# B&R Automation Studio project Parker_BMM_ST_V5_3147_V12 (part 17)

#### cur_draw.c
```c
/********************************************************************
 * COPYRIGHT --  B&R CHINA
 ********************************************************************
 * Program: cur_draw
 * File: cur_draw.c
 * Author: lijianjun
 * Created: March 06, 2013
 ********************************************************************
 * Implementation of program cur_draw --- thick profile curve draw in HMI
 ********************************************************************/

#include <bur/plctypes.h>
#include <string.h>

#ifdef _DEFAULT_INCLUDES
#include <AsDefault.h>
#endif

/***********************************************************************************
** 			                    Include user files								  **
***********************************************************************************/
#include "draw.h"
#include "pic_id.h"
#include "thick.h"

/***********************************************************************************
                             Function Declarations
***********************************************************************************/
UINT vsLine( UDINT VCHandle, UINT x1, UINT y1,UINT x2, UINT y2, USINT color);
UINT vsLineH( UDINT VCHandle, UINT x, UINT y, UINT len, USINT color);
UINT vsLineV( UDINT VCHandle, UINT x, UINT y, UINT len, USINT color);
UINT vsRect(  UDINT VCHandle, UINT x1, UINT y1,UINT x2, UINT y2, USINT color);

/**********************************************************************************
**     	        		 I N I T U P  O F   T H E   T A S K 		 		     **
**********************************************************************************/
_INIT  void init(void)
{
	width 		= 	VSCREEN_WIDTH;
	height 		= 	VSCREEN_HEIGHT;
	backColor  	= 	VSCREEN_COLOR_BACKGROUND;
	frameColor 	= 	VSCREEN_COLOR_FRAME;
	crossColor	= 	VSCREEN_COLOR_CROSS_CURSOR;
	fillColor   =  VSCREEN_COLOR_BACKGROUND;

	ORIGINAL_X0  = 100;
	ORIGINAL_Y0  = 150;

	rSetScale = 0.1;
	rActScale = 1.0;
	xScaleBmp = 0;

	drawStep = 0;
}/*  end of INIT */

/**********************************************************************************
**        	     C Y C L I C   P A R T   O F   T H E   T A S K  				 **
**********************************************************************************/
_CYCLIC void cyc(void)
{
	INT X,Y;

	if((gPanelObj.GetPicture == PIC_CURVE_TRACE) ||
		(1 == gThickProf.FunOption.IsTraceInEdit && gPanelObj.GetPicture == PIC_CURVE_EDIT))
	{
		if (memcmp(getAT,gThickData.RealData,sizeof(getAT)) != 0 && DrawMan.draw == 0)
		{
			DrawMan.draw = 1;
			memcpy(getAT,gThickData.RealData,sizeof(getAT));
		}
	}

	if (gPanelObj.GetPicture == PIC_CURVE_EDIT)
	{
		if (DRAW_PIC != PIC_CURVE_EDIT && DRAW_PIC != 255)
		{
			DrawMan.draw = 1;
		}
		DRAW_PIC = PIC_CURVE_EDIT;
	}
	else if (gPanelObj.GetPicture == PIC_CURVE_TRACE)
	{
		if (DRAW_PIC != PIC_CURVE_TRACE && DRAW_PIC != 255)
		{
			DrawMan.draw = 1;
		}
		DRAW_PIC = PIC_CURVE_TRACE;
	}
	else
	{
		DRAW_PIC = 255;
	}

	if (gPanelObj.GetPicture == PIC_CURVE_EDIT || gPanelObj.GetPicture == PIC_CURVE_TRACE)
	{
		switch (drawStep)
		{
			case 0:
				vcHandle = VA_Setup(1,gPanelObj.VisualName);
				if (vcHandle)  drawStep = 100;
				break;

			case 100:
				status = VA_Saccess(1, vcHandle);
				if(status == 0)
				{
					drawStep = 200;
				}
				break;

			case 200:
				Status_Attach = 1;
				if (gPanelObj.GetPicture == PIC_CURVE_EDIT)
				{
					Status_Attach = VA_Attach(1,vcHandle,0,(UDINT)"Page_82_Profile/Default/DrawBox_1");
				}
				else
				{
					Status_Attach = VA_Attach(1,vcHandle,0,(UDINT)"Page_83_Trace/Default/DrawBox_1");
				}
				if(Status_Attach == 0)
				{
					/* Get width of DrawBox Control*/
					VA_GetDisplayInfo(1,vcHandle,1,(UDINT)&Drawbox_width);
					/* Get height of DrawBox Control */
					VA_GetDisplayInfo(1,vcHandle,2,(UDINT)&Drawbox_height);

					drawStep = 300;
				}
				else
				{
					VA_Srelease(1, vcHandle);
					drawStep = 100;
				}
				break;
			case 300:
				xMax = 0.0;
				for(i=0;i<= S$THICK_MAX;i++)
					{
					if(xMax < SetPos[i].x)xMax = SetPos[i].x;
				}

				if (usScaleIndex == 1) //ipis0619
				{
					rSetScale = 0.4;
					rActScale = 4.0;
					xScaleBmp = 2;
				}else if (usScaleIndex == 2)
				{
					rSetScale = 0.2;
					rActScale = 2.0;
					xScaleBmp = 1;
				}else
				{
					rSetScale = 0.1;
					rActScale = 1.0;
					xScaleBmp = 0;
				}
		/*---//ipis0619 -----------------------------------------*/
//				if(xMax >= 1500)
//				{
//					rSetScale = 0.1;
//					rActScale = 1.0;
//					xScaleBmp = 0;
//				}
//				else if(xMax >= 750)
//				{
//					rSetScale = 0.2;
//					rActScale = 2.0;
//					xScaleBmp = 1;
//				}
//				else
//				{
//					rSetScale = 0.4;
//					rActScale = 4.0;
//					xScaleBmp = 2;
//				}
		/*---//ipis0619 -----------------------------------------*/
				status = VA_Redraw (1,vcHandle);
				if(0 == status)
				{
					if (gPanelObj.GetPicture == PIC_CURVE_EDIT)  drawStep  = 400;
					if (gPanelObj.GetPicture == PIC_CURVE_TRACE) drawStep  = 600;
				}
				break;
			/**************draw the setting curve*************/
			case 400:
				for(i=0;i<= S$THICK_MAX;i++)
					{
					X = (INT)(SetPos[i].x*rSetScale + 0.1);
					if(X > Drawbox_width - 2)X = Drawbox_width - 2;
					Y = S$THICK_POINT - SetPos[i].y;    /* 0 <SetPos[i].y <= 399  ->  1 < Y < 400*/

					vsLineH(vcHandle,0,Y,Drawbox_width-1,VSCREEN_COLOR_BACKGROUND);

					if (1 == CurveNode[i].flagNode)
					{
						if(i == DrawMan.currentNode && 1 == DrawMan.flagLineFocus)
						{
							vsLineH(vcHandle,0,Y,X,crossColor);
							vsLineH(vcHandle,0,Y,DrawMan.weight*rSetScale,VSCREEN_COLOR_WEIGHT);
						}
						else
						{
							vsLineH(vcHandle,0,Y,X,VSCREEN_COLOR_CURVE);
							vsLineH(vcHandle,0,Y,DrawMan.weight*rSetScale,VSCREEN_COLOR_WEIGHT);
						}
					}
					else
					{
						vsLineH(vcHandle,0,Y,X,VSCREEN_COLOR_UNFOCUS_LINE);
						vsLineH(vcHandle,0,Y,DrawMan.weight*rSetScale,VSCREEN_COLOR_WEIGHT);
					}

					if(0 == DrawMan.flagLineFocus)
					{
						if(i > CurveNode[DrawMan.currentNode].former + 1 && i <= DrawMan.currentNode)
						{
							vsLine(vcHandle,(INT)(SetPos[i-1].x*rSetScale + 0.1),S$THICK_POINT - SetPos[i-1].y,X,Y,crossColor);
								}
						else
						{
							if(i > 0)
							{
								vsLine(vcHandle,(INT)(SetPos[i-1].x*rSetScale + 0.1),S$THICK_POINT - SetPos[i-1].y,X,Y,VSCREEN_COLOR_CURVE);
									}
						}
					}
					else
					{
						if(i > 0)
						{
							vsLine(vcHandle,(INT)(SetPos[i-1].x*rSetScale + 0.1),S$THICK_POINT - SetPos[i-1].y,X,Y,VSCREEN_COLOR_CURVE);
								}
					}
				}

				if(DrawMan.step == S$STEP_ADDLINE)
					{
					drawStep = 500;
				}
				else
				{
					drawStep = 550;
				}
				break;
			/*---draw the cross line ---*/
			case 500:
				xTemp = (INT)(SetPos[DrawMan.currentPoint].x*rSetScale + 0.1) - 20;
				if(xTemp < 0)xTemp = 0;

				if(xTemp + 40 < width)
				{
					xLength = 40;
				}
				else
				{
					xLength = width - 40;
				}
				vsLineH(vcHandle,xTemp,S$THICK_POINT - DrawMan.currentPoint,xLength,crossColor);

					yTemp	= S$THICK_POINT - DrawMan.currentPoint - 20;
				if(yTemp < 0)yTemp = 0;

				if(yTemp + 40 < height)
				{
					yLength = 40;
				}
				else
				{
					yLength = height - 40;
				}
				vsLineV(vcHandle,(INT)(SetPos[DrawMan.currentPoint].x*rSetScale + 0.1),yTemp,yLength,crossColor);
				drawStep = 550;
				break;
			/*------ is or not draw the trace curve in edit profile page ------*/
			case 550:
				if(1 == gThickProf.FunOption.IsTraceInEdit)
				{
					drawStep = 700;
				}
				else
				{
					drawStep = 900;
				}
				break;
			/**************draw the setting curve*************/
			case 600:
				for(i=0;i<= S$THICK_MAX;i++)
					{
					vsLineH(vcHandle,0,S$THICK_POINT - SetPos[i].y,Drawbox_width-1,VSCREEN_COLOR_BACKGROUND);
						vsLineH(vcHandle,0,S$THICK_POINT - SetPos[i].y,(INT)(SetPos[i].x*rSetScale + 0.1),VSCREEN_COLOR_UNFOCUS_LINE);
						}
				drawStep = 700;
				break;
			/**************draw the trace curve*************/
			case 700:
				for(i=0;i<S$THICK_SAMPLE-1;i++)
					{
					if (getAT[i+1] != 0)
					{
						firstPos.x  = getAT[i] * rActScale;
						firstPos.y  = i*4;
						secondPos.x = getAT[i+1] * rActScale;
						secondPos.y = (i+1)*4;
						status = vsLine(vcHandle, firstPos.x, S$THICK_POINT-firstPos.y, secondPos.x, S$THICK_POINT-secondPos.y, crossColor);
							}
				}

				if(getAT[S$THICK_SAMPLE-1]!= 0)
					{
					status = vsLine(vcHandle, getAT[S$THICK_SAMPLE-1] * rActScale, S$THICK_POINT - 396, getAT[S$THICK_SAMPLE-1] * rActScale, S$THICK_POINT - 399, crossColor);
						}
				drawStep = 900;
				break;
			/* copy the screen to interface  */
			case 900:
				vsRect(vcHandle,0,0,VSCREEN_WIDTH-1,VSCREEN_HEIGHT-1,VSCREEN_COLOR_FRAME);
				VA_Redraw (1,vcHandle);
				VA_Detach(1,vcHandle);
				VA_Srelease(1, vcHandle);
				if((gPanelObj.GetPicture == PIC_CURVE_EDIT) || (gPanelObj.GetPicture == PIC_CURVE_TRACE))
				{
					DrawMan.draw = 0;
					drawStep = 1000;
				}
				else
				{
					drawStep = 2000;
				}
				break;
			/*	waiting for draw  */
			case 1000:
				if (1 == DrawMan.draw )
				{
					drawStep  = 100;
				}
				break;
			case 2000:
				drawStep  = 100;
				break;
		}
	}
	else
	{
		if (drawStep != 0 && vcHandle != 0) drawStep = 100;
	}

}/*end of CYCLIC*/

UINT vsLine( UDINT VCHandle, UINT x1, UINT y1,UINT x2, UINT y2, USINT color)
{
	if(x1 > Drawbox_width-2)x1 = Drawbox_width-2;
	if(x2 > Drawbox_width-2)x2 = Drawbox_width-2;
	return  VA_Line(1, VCHandle,x1,y1,x2,y2,color);
}

UINT vsLineH( UDINT VCHandle, UINT x, UINT y, UINT len, USINT color)
{
	if(x+len <= Drawbox_width-2)
	{
		return  VA_Line(1, VCHandle,x,y,x+len,y,color);
	}
	else
	{
		return  VA_Line(1, VCHandle,x,y,Drawbox_width-2,y,color);
	}
}

UINT vsLineV( UDINT VCHandle, UINT x, UINT y, UINT len, USINT color)
{
	if(x > Drawbox_width-2)x = Drawbox_width-2;
	return  VA_Line(1, VCHandle,x,y,x,y+len,color);
}

UINT vsRect(  UDINT VCHandle, UINT x1, UINT y1,UINT x2, UINT y2, USINT color)
{
	return VA_Rect(1,VCHandle,x1,y1,x2-x1,y2-y1,255,color);
}
```

#### cur_draw.var
```iecst
VAR
	vcHandle : UDINT;
	xTemp : INT;
	xLength : INT;
	yTemp : INT;
	yLength : INT;
	width : UINT;
	Drawbox_width : UDINT;
	Drawbox_height : UDINT;
	height : UINT;
	backColor : UINT;
	fillColor : UINT;
	frameColor : UINT;
	crossColor : UINT;
	xMax : INT;
	xScaleBmp : UINT;
	rSetScale : REAL;
	rActScale : REAL;
	status : UINT;
	Status_Attach : UINT;
	drawStep : UINT;
	i : UINT;
	getAT : ARRAY[0..99] OF INT;
	DRAW_PIC : UINT;
	firstPos : position_typ;
	secondPos : position_typ;
END_VAR
```

### Program Logical/thickness/cur_edit (ANSIC, version 1.00.0) - profile edit

#### cur_edit.c
```c
/********************************************************************
 * COPYRIGHT --  B&R CHINA
 ********************************************************************
 * Program: cur_edit
 * File: cur_edit.c
 * Author: lijianjun
 * Created: March 06, 2013
 ********************************************************************
 * Implementation of program cur_edit --- thick profile curve data compiling
 ********************************************************************/

#include <bur/plctypes.h>
#include <string.h>

#ifdef _DEFAULT_INCLUDES
#include <AsDefault.h>
#endif

/***********************************************************************************
** 					 	        Include user files								             **
***********************************************************************************/
#include "keyap2100.h"
#include "pic_id.h"
#include "draw.h"
#include "thick.h"
#include "edge.h"               /*edge function
/**********************************************************************************
**                            Function Declarations								      **
**********************************************************************************/
void nodeAdd(USINT *enable,UINT nodeNum); /*insert a horizontal line*/
void nodeDel(USINT *enable,UINT nodeNum); /*delete a horizontal line*/
void curveScan(SINT *upDown);  			   /*scan the horizontal to get the focus*/
void curveQuickScan(SINT *upDown);  		/*scan the horizontal to get the focus*/
void curveColor(USINT *action);			   /* */
void vxEdit();
void vxEditUnit(INT unitLength);
void moveCross(SINT *upDown);
void weightSet();
void curveToLine(USINT *action,UINT nodeNum);
void curveMove();
void curveClear();
/**********************************************************************************
**     	        	 I N I T U P  O F   T H E   T A S K 		 				 **
**********************************************************************************/
_INIT  void init(void)
{
	RTInfo_v.enable = 1;
	RTInfo(&RTInfo_v);
	TimeLenth = RTInfo_v.cycle_time/4000;
	tTask = RTInfo_v.cycle_time/1000.0/1000.0;

	TimeLenth  = TimeLenth /6 * 6;
	StepLength = TimeLenth;

	focusColor 		= VSCREEN_COLOR_FOCUS_LINE;
	unfocusColor 	= VSCREEN_COLOR_UNFOCUS_LINE;

	addNode 		= 0;
	delNode 		= 0;
	scanNode  	= 0;
	scanLine    = 0;
	setColor		= 0;
	isDownLoad  = 0;

	memset(oldSetPos,0,sizeof(oldSetPos));
	DrawMan.step  = S$STEP_EDIT;
	DrawMan.input = 0;

	Counter = 0;
	CurevInitDownload = 1;

	moveValue = 0;
	bBackEnable = 0;
	bRedoEnable = 0;

	memset(&gThickProf.IsMarker[0],0,sizeof(gThickProf.IsMarker));
	memset(&IsMarkerOld[0],0,sizeof(IsMarkerOld));

	MarkPercentOld = MarkPercent = 20;

	bStartUpLineFocus = 0;
	bStartDnLineFocus = 0;
	cntUpButtonPress = 0;
	cntDownButtonPress = 0;
}/*  end of init   */
/**********************************************************************************
**            C Y C L I C   P A R T   O F   T H E   T A S K  				     **
**********************************************************************************/
_CYCLIC void cyc(void)
{
	if(1 == gRecipeOperate.OnceOk && 1 == gRecipeOperate.CurveOk)
	{
		if(1 == CurevInitDownload)
		{
			CurevInitDownload = 0;
			DrawMan.downLoad  = 1;
		}

		if(1 == GapMaxLimitChange)
		{
			GapMaxLimitChange = 0;
			DrawMan.downLoad  = 1;
		}
	}

	/*IsZeroDn Change */
	if(IsZeroDnOld != gThickProf.FunOption.IsZeroDn)
	{
		DrawMan.downLoad = 1;
	}

	IsZeroDnOld = gThickProf.FunOption.IsZeroDn;

	/*  mark point --- display  */
	if((PIC_MARKER_SET_A == GetPictureOld) && (gPanelObj.GetPicture != PIC_MARKER_SET_A))
	{
		memset(&gThickProf.IsMarker[0],0,sizeof(gThickProf.IsMarker));
		memset(&IsMarkerOld[0],0,sizeof(IsMarkerOld));
		DrawMan.downLoad = 1;
	}
	GetPictureOld = gPanelObj.GetPicture;

	if(MarkPercent < -50 || MarkPercent > 50)MarkPercent = 20;
	if(MarkPercentOld != MarkPercent)
	{
		DrawMan.downLoad = 1;
	}
	MarkPercentOld = MarkPercent;

	if (memcmp(gThickProf.IsMarker,IsMarkerOld,sizeof(IsMarkerOld)) != 0)
	{
		memcpy(IsMarkerOld,gThickProf.IsMarker,sizeof(gThickProf.IsMarker));
		DrawMan.downLoad = 1;
	}

	if(ServoMinOld != gThickData.ServoMin)
	{
		isDownLoad = 2;
	}

	ServoMinOld = gThickData.ServoMin;

	if(ServoMaxOld != gThickData.ServoMax)
	{
		isDownLoad = 2;
	}

	ServoMaxOld = gThickData.ServoMax;

	if (1 == DrawMan.downLoad)
	{
		for (i = 0; i< 100; i++)
		{
			if(gMachineFix.Parison.eActuatorType == ACTUATOR_ELECTRIC  || 0 == gThickData.IsZeroDn)
			{
				gThickData.SetData[i] = gThickData.ServoMin + gThickData.ServoLength * (SetPos[i*4].x +
					SetPos[i*4+1].x + SetPos[i*4+2].x + SetPos[i*4+3].x)/12000;

				if(1 == gThickProf.IsMarker[i])
				{
					if(0 == i)
					{
						gThickData.SetData[i] = gThickData.SetData[i] + gThickData.ServoLength * MarkPercent / 100;
						if(gThickData.SetData[i] < gThickData.ServoMin)gThickData.SetData[i] = gThickData.ServoMin;
						if(gThickData.SetData[i] > gThickData.ServoMax)gThickData.SetData[i] = gThickData.ServoMax;

						gThickData.SetData[i+1] = gThickData.SetData[i+1] + gThickData.ServoLength * MarkPercent / 200;
						if(gThickData.SetData[i+1] < gThickData.ServoMin)gThickData.SetData[i+1] = gThickData.ServoMin;
						if(gThickData.SetData[i+1] > gThickData.ServoMax)gThickData.SetData[i+1] = gThickData.ServoMax;

					}
					else if(99 == i)
					{
						gThickData.SetData[i-1] = gThickData.SetData[i-1] + gThickData.ServoLength * MarkPercent / 200;
						if(gThickData.SetData[i-1] < gThickData.ServoMin)gThickData.SetData[i-1] = gThickData.ServoMin;
						if(gThickData.SetData[i-1] > gThickData.ServoMax)gThickData.SetData[i-1] = gThickData.ServoMax;

						gThickData.SetData[i] = gThickData.SetData[i] + gThickData.ServoLength * MarkPercent / 100;
						if(gThickData.SetData[i] < gThickData.ServoMin)gThickData.SetData[i] = gThickData.ServoMin;
						if(gThickData.SetData[i] > gThickData.ServoMax)gThickData.SetData[i] = gThickData.ServoMax;
					}
					else
					{
						gThickData.SetData[i-1] = gThickData.SetData[i-1] + gThickData.ServoLength * MarkPercent / 200;
						if(gThickData.SetData[i-1] < gThickData.ServoMin)gThickData.SetData[i-1] = gThickData.ServoMin;
						if(gThickData.SetData[i-1] > gThickData.ServoMax)gThickData.SetData[i-1] = gThickData.ServoMax;

						gThickData.SetData[i] = gThickData.SetData[i] + gThickData.ServoLength * MarkPercent / 100;
						if(gThickData.SetData[i] < gThickData.ServoMin)gThickData.SetData[i] = gThickData.ServoMin;
						if(gThickData.SetData[i] > gThickData.ServoMax)gThickData.SetData[i] = gThickData.ServoMax;

						gThickData.SetData[i+1] = gThickData.SetData[i+1] + gThickData.ServoLength * MarkPercent / 200;
						if(gThickData.SetData[i+1] < gThickData.ServoMin)gThickData.SetData[i+1] = gThickData.ServoMin;
						if(gThickData.SetData[i+1] > gThickData.ServoMax)gThickData.SetData[i+1] = gThickData.ServoMax;
					}
				}
			}
			else if( gMachineFix.Parison.eActuatorType == ACTUATOR_HYD && 1 == gThickData.IsZeroDn)
			{
				gThickData.SetData[i] = gThickData.ServoMax - gThickData.ServoLength * (SetPos[i*4].x +
					SetPos[i*4+1].x + SetPos[i*4+2].x + + SetPos[i*4+3].x)/12000;

				if(1 == gThickProf.IsMarker[i])
				{
					if(0 == i)
					{
						gThickData.SetData[i] = gThickData.SetData[i] - gThickData.ServoLength * MarkPercent / 100;
						if(gThickData.SetData[i] < gThickData.ServoMin)gThickData.SetData[i] = gThickData.ServoMin;
						if(gThickData.SetData[i] > gThickData.ServoMax)gThickData.SetData[i] = gThickData.ServoMax;

						gThickData.SetData[i+1] = gThickData.SetData[i+1] - gThickData.ServoLength * MarkPercent / 200;
						if(gThickData.SetData[i+1] < gThickData.ServoMin)gThickData.SetData[i+1] = gThickData.ServoMin;
						if(gThickData.SetData[i+1] > gThickData.ServoMax)gThickData.SetData[i+1] = gThickData.ServoMax;
					}
					else if(99 == i)
					{
						gThickData.SetData[i-1] = gThickData.SetData[i-1] - gThickData.ServoLength * MarkPercent / 200;
						if(gThickData.SetData[i-1] < gThickData.ServoMin)gThickData.SetData[i-1] = gThickData.ServoMin;
						if(gThickData.SetData[i-1] > gThickData.ServoMax)gThickData.SetData[i-1] = gThickData.ServoMax;

						gThickData.SetData[i] = gThickData.SetData[i] - gThickData.ServoLength * MarkPercent / 100;
						if(gThickData.SetData[i] < gThickData.ServoMin)gThickData.SetData[i] = gThickData.ServoMin;
						if(gThickData.SetData[i] > gThickData.ServoMax)gThickData.SetData[i] = gThickData.ServoMax;
					}
					else
					{
						gThickData.SetData[i-1] = gThickData.SetData[i-1] - gThickData.ServoLength * MarkPercent / 200;
						if(gThickData.SetData[i-1] < gThickData.ServoMin)gThickData.SetData[i-1] = gThickData.ServoMin;
						if(gThickData.SetData[i-1] > gThickData.ServoMax)gThickData.SetData[i-1] = gThickData.ServoMax;

						gThickData.SetData[i] = gThickData.SetData[i] - gThickData.ServoLength * MarkPercent / 100;
						if(gThickData.SetData[i] < gThickData.ServoMin)gThickData.SetData[i] = gThickData.ServoMin;
						if(gThickData.SetData[i] > gThickData.ServoMax)gThickData.SetData[i] = gThickData.ServoMax;

						gThickData.SetData[i+1] = gThickData.SetData[i+1] - gThickData.ServoLength * MarkPercent / 200;
						if(gThickData.SetData[i+1] < gThickData.ServoMin)gThickData.SetData[i+1] = gThickData.ServoMin;
						if(gThickData.SetData[i+1] > gThickData.ServoMax)gThickData.SetData[i+1] = gThickData.ServoMax;
					}
				}
			}

			x_Profile[i] = (SetPos[i*4].x + SetPos[i*4+1].x + SetPos[i*4+2].x + SetPos[i*4+3].x)/120.0;
		}

		memcpy(oldSetPos,SetPos,sizeof(SetPos));

		DrawMan.downLoad  		 = 0;
		gRecipeOperate.CurveSave = 1;
		isDownLoad        		 = 0;

	}/* if (1 == DrawMan.downLoad) */

	if(gPanelObj.GetPicture == PIC_CURVE_EDIT)
	{
		gPanelObj.LedMatric[S$KEYMATRIX_F15] =  0;
		gPanelObj.LedMatric[S$KEYMATRIX_F15] = isDownLoad;
	}
	else if(gPanelObj.GetPicture == PIC_THICK_START)
	{
		gPanelObj.LedMatric[S$KEYMATRIX_F15] = isDownLoad;
		gPanelObj.LedMatric[S$KEYMATRIX_F15] =  0;
	}
	else
	{
		gPanelObj.LedMatric[S$KEYMATRIX_F15] =  0;
		gPanelObj.LedMatric[S$KEYMATRIX_F15] =  0;
	}

	if(gPanelObj.GetPicture != PIC_CURVE_EDIT  && gPanelObj.GetPicture != PIC_THICK_START)
	{
		Counter = 0;
		return;
	}

	Counter ++;
	if(Counter > 1000)Counter = 120;
	if(Counter < 15)return;

	if(0 == gThickProf.FunOption.IsAccu)
	{
		AccuColor  = 0x0060;
		ContiColor = 0x003A;

	}
	else
	{
		AccuColor  = 0x003A;
		ContiColor = 0x0060;
	}

	if((gPanelObj.PasswordLevel >= 1)&&(1 == DrawMan.flagLineFocus)&& (DrawMan.step == S$STEP_EDIT))
	{
		inputenable = 1;
	}
	else
	{
		inputenable = 0;
	}

	bHideBack = ! bBackEnable;

	if(gPanelObj.GetPicture == PIC_CURVE_EDIT)
	{
		if(gPanelObj.PasswordLevel >= 1)
		{
			if(gPanelObj.PasswordLevel >= 3)
			{
			//	changeButton = gPanelObj.KeyMatric[S$KEYMATRIX_F7];
			}
			else
			{
				changeButton = 0;
			}
//			delButton 		= gPanelObj.KeyMatric[S$KEYMATRIX_F8] | gPanelObj.KeyMatric[S$KEYMATRIX_DEL];
//			curtolButton 	= gPanelObj.KeyMatric[S$KEYMATRIX_F9] | bCurveChangeLine;
			delButton 		=  gPanelObj.KeyMatric[S$KEYMATRIX_DEL];
			curtolButton 	=  bCurveChangeLine;
			escButton 		= gPanelObj.KeyMatric[S$KEYMATRIX_ESC];
			downloadButton	= gPanelObj.KeyMatric[S$KEYMATRIX_F15];

//			v1Add 			= gPanelObj.KeyMatric[S$KEYMATRIX_F13] | bCurveDnRight;
//			v1Sub 			= gPanelObj.KeyMatric[S$KEYMATRIX_F12] | bCurveDnLeft;
//			v2Add 			= gPanelObj.KeyMatric[S$KEYMATRIX_F11] | bCurveUpRight;
//			v2Sub 			= gPanelObj.KeyMatric[S$KEYMATRIX_F10] | bCurveUpLeft;
				v1Add 			=  bCurveDnRight;
				v1Sub 			=  bCurveDnLeft;
				v2Add 			= bCurveUpRight;
				v2Sub 			=  bCurveUpLeft;
			v03Sub 		   = gPanelObj.KeyMatric[S$KEYMATRIX_LEFT];
			v03Add 		   = gPanelObj.KeyMatric[S$KEYMATRIX_RIGHT];

			weightUpButton   = bWeightUp;
			weightDownButton = bWeightDown;

			if(1 == gPanelObj.KeyMatric[S$KEYMATRIX_UP])
			{
			/*-//ipis0619--------------------------------------------------------------------------------*/
//				cntUpButtonPress = cntUpButtonPress + 1;
//				if(cntUpButtonPress >= 10000)cntUpButtonPress = 100;
//
//				if((cntUpButtonPress % 12) < 8)
//				{
//					upButton = 1;
//				}
//				else
//				{
//					upButton = 0;
//				}
			/*-//ipis0619--------------------------------------------------------------------------------*/
			upButton = 1;	 //ipis0619
			}
			else
			{
				cntUpButtonPress = 0;
				upButton = 0;
			}

			if(1 == gPanelObj.KeyMatric[S$KEYMATRIX_DOWN])
			{
			/*-//ipis0619--------------------------------------------------------------------------------*/
//				cntDownButtonPress = cntDownButtonPress + 1;
//				if(cntDownButtonPress >= 10000)cntDownButtonPress = 100;
//
//				if((cntDownButtonPress % 12) < 8)
//				{
//					downButton = 1;
//				}
//				else
//				{
//					downButton = 0;
//				}
			/*-//ipis0619--------------------------------------------------------------------------------*/
			downButton = 1;	//ipis0619
			}
			else
			{
				cntDownButtonPress = 0;
				downButton = 0;
			}

			if(1 == bQuickUp)
			{
			/*-//ipis0619--------------------------------------------------------------------------------*/
//				cntQuickUpPress = cntQuickUpPress + 1;
//				if(cntQuickUpPress >= 12000)cntQuickUpPress = 120;
//
//				if((cntQuickUpPress % 12) < 8)
//				{
//					quickUpButton = 1;
//				}
//				else
//				{
//					quickUpButton = 0;
//				}
			/*-//ipis0619--------------------------------------------------------------------------------*/
			quickUpButton = 1;	//ipis0619
			}
			else
			{
				cntQuickUpPress = 0;
				quickUpButton = 0;
			}

			if(1 == bQuickDown)
			{
			/*-//ipis0619--------------------------------------------------------------------------------*/
//				cntQuickDownPress = cntQuickDownPress + 1;
//				if(cntQuickDownPress >= 12000)cntQuickDownPress = 120;
//
//				if((cntQuickDownPress % 12) < 8)
//				{
//					quickDownButton = 1;
//				}
//				else
//				{
//					quickDownButton = 0;
//				}
			/*-//ipis0619--------------------------------------------------------------------------------*/
				quickDownButton = 1;
			}
			else
			{
				cntQuickDownPress = 0;
				quickDownButton = 0;
			}

			if(1 == bFocusUp)
			{
		/*-//ipis0619--------------------------------------------------------------------------------*/
//				cntFocusUpPress = cntFocusUpPress + 1;
//				if(cntFocusUpPress >= 7000)cntFocusUpPress = 700;
//
//				if((cntFocusUpPress % 7) < 4)
//				{
//					focusUpButton = 1;
//				}
//				else
//				{
//					focusUpButton = 0;
//				}
		/*-//ipis0619--------------------------------------------------------------------------------*/
			focusUpButton = 1;
			}
			else
			{
				cntFocusUpPress = 0;
				focusUpButton = 0;
			}

			if(1 == bFocusDown)
			{
		/*-//ipis0619--------------------------------------------------------------------------------*/
//				cntFocusDownPress = cntFocusDownPress + 1;
//				if(cntFocusDownPress >= 7000)cntFocusDownPress = 700;
//
//				if((cntFocusDownPress % 7) < 4)
//				{
//					focusDownButton = 1;
//				}
//				else
//				{
//					focusDownButton = 0;
//				}
		/*-//ipis0619--------------------------------------------------------------------------------*/
				focusDownButton = 1;
			}
			else
			{
				cntFocusDownPress = 0;
				focusDownButton = 0;
			}

			tabButton = gPanelObj.KeyMatric[S$KEYMATRIX_TAB];

			if(1 == bCurveInit)
			{
				cntPressbuttonTime = cntPressbuttonTime + 1;
			}
			else
			{
				cntPressbuttonTime = 0;
			}

			if( cntPressbuttonTime * TimeLenth * 4 > 3000)
			{
				clearButton = 1;
			}
			else
			{
				clearButton = 0;
			}
		}
		else
		{
//			if(1 == gPanelObj.KeyMatric[S$KEYMATRIX_DOWN] ||
//				1 == gPanelObj.KeyMatric[S$KEYMATRIX_UP]   ||
//				1 == gPanelObj.KeyMatric[S$KEYMATRIX_LEFT] ||
//				1 == gPanelObj.KeyMatric[S$KEYMATRIX_RIGHT]||
//				1 == gPanelObj.KeyMatric[S$KEYMATRIX_F7]   ||
//				1 == gPanelObj.KeyMatric[S$KEYMATRIX_F8]   ||
//				1 == gPanelObj.KeyMatric[S$KEYMATRIX_F9]   ||
//				1 == gPanelObj.KeyMatric[S$KEYMATRIX_F10]  ||
//				1 == gPanelObj.KeyMatric[S$KEYMATRIX_F11]  ||
//				1 == gPanelObj.KeyMatric[S$KEYMATRIX_F12]  ||
//				1 == gPanelObj.KeyMatric[S$KEYMATRIX_F13]  ||
//				1 == gPanelObj.KeyMatric[S$KEYMATRIX_ESC]  ||
//				1 == gPanelObj.KeyMatric[S$KEYMATRIX_DEL])
//				{
//				gImply.PsdLevel1 = 1;
//			}
//
//			downloadButton	= gPanelObj.KeyMatric[S$KEYMATRIX_F15];
//			cntUpButtonPress   = 0;
//			cntDownButtonPress = 0;
//			cntQuickUpPress = 0;
//			cntQuickDownPress = 0;
//			cntFocusUpPress = 0;
//			cntFocusDownPress = 0;
		}
	}
	else if(gPanelObj.GetPicture == PIC_THICK_START)
	{
		downloadButton	= gPanelObj.KeyMatric[S$KEYMATRIX_F15];
	}

	R_TRIG_DOWNLOAD.CLK = downloadButton;
	R_TRIG(&R_TRIG_DOWNLOAD);
	if (1 == R_TRIG_DOWNLOAD.Q)
	{
		DrawMan.downLoad = 1;
	}

	if (memcmp(SetPos,oldSetPos,sizeof(SetPos)) != 0)
	{
		memcpy(oldSetPos,SetPos,sizeof(SetPos));
		DrawMan.draw = 1;
		isDownLoad   = 2;
	}

	if (inputok == 0)
	{
		currentGap = SetPos[tempIndex % S$THICK_POINT].x;
		oldcurrentGap = currentGap;
	}

	if(0 == gThickProf.FunOption.Is100_300)
	{
		currentIndex = tempIndex;
	}
	else
	{
		currentIndex = tempIndex/4;
	}

	if(1 == gThickProf.FunOption.Is100_300)
	{
		IndexAddLineMax = 99;
		if(IndexAddLine > 99)IndexAddLine = 99;
	}
	else
	{
		IndexAddLineMax = 399;
		if(IndexAddLine > 399)IndexAddLine = 399;
	}

	switch (DrawMan.step)
	{
		case S$STEP_EDIT:
			if(0 == gThickProf.FunOption.bLengthUnit)
			{
				vxEdit();
			}
			else
			{
				if(LengthUnit < 3)LengthUnit = 3;
				if(LengthUnit > 150)LengthUnit = 150;
				vxEditUnit(LengthUnit);
			}

			tempIndex = DrawMan.currentNode;

			if(gPanelObj.PasswordLevel >= 2)  //ipis0619
			{
			moveInputEnable = 1;
			}
			else
			{
			moveInputEnable = 0;
			}

			if(1 == moveInputOk)
			{
				moveInputOk = 0;
				if(moveValue != 0)
				{
					bBackEnable = 1;
					memcpy(&mDrawMan,&DrawMan,sizeof(mDrawMan));
					memcpy(&mCurveNode,&CurveNode,sizeof(mCurveNode));
					memcpy(&mSetPos,&SetPos,sizeof(mSetPos));
					DrawMan.step = S$STEP_CURVEMOVE;
				}
			}

			if(1 == bBackEnable && 1 == bKeyBack)
			{
				bBackEnable = 0;
				DrawMan.step = S$STEP_UNDO;
			}

			if(1 == bRedoEnable && 1 == bKeyRedo)
			{
				bRedoEnable = 0;
				DrawMan.step = S$STEP_REDO;
			}

			R_TRIG_UP.CLK = upButton;
			R_TRIG(&R_TRIG_UP);
			R_TRIG_DOWN.CLK = downButton;
			R_TRIG(&R_TRIG_DOWN);

			if ( R_TRIG_UP.Q == 1)   scanNode = 1;
			if ( R_TRIG_DOWN.Q == 1) scanNode = -1;

			R_TRIG_QUICK_UP.CLK = 	quickUpButton;
			R_TRIG(&R_TRIG_QUICK_UP);
			R_TRIG_QUICK_DOWN.CLK = quickDownButton;
			R_TRIG(&R_TRIG_QUICK_DOWN);

			if ( R_TRIG_QUICK_UP.Q == 1)   scanLine = 1;
			if ( R_TRIG_QUICK_DOWN.Q == 1) scanLine = -1;

			if(1 == bAddLineMode)
			{
				bAddLineMode = 0;
				if(1 == gThickProf.FunOption.Is100_300)
				{
					if(0 == IndexAddLine)IndexAddLine = DrawMan.currentNode;
					DrawMan.currentPoint = IndexAddLine * 4;
				}
				else
				{
					if(0 == IndexAddLine)IndexAddLine = DrawMan.currentNode;
					DrawMan.currentPoint = IndexAddLine;
				}
				DrawMan.step  = S$STEP_ADDLINE;
				setColor = 2;
				IndexAddLine = 0;
			}

			if(1 == focusUpButton || 1 == focusDownButton)
			{
				DrawMan.currentPoint = DrawMan.currentNode;;
				DrawMan.step = S$STEP_ADDLINE;
				setColor = 2;
			}

			if(0 == gPanelObj.vcHandle)
			{
				gPanelObj.vcHandle = VA_Setup(1, gPanelObj.VisualName);
			}

			if (gPanelObj.vcHandle != 0)
			{
				if (!VA_Saccess(1, gPanelObj.vcHandle))
				{
					VA_GetTouchAction (1,gPanelObj.vcHandle,0,(UDINT)(&TouchPoint));
					VA_Srelease(1, gPanelObj.vcHandle);
				}
			}

			if(1 == TouchPoint.status)
			{
				cntPressed = cntPressed + 1;

				if(10 == cntPressed)
				{
					if(TouchPoint.x > ORIGINAL_X0 + 10 && TouchPoint.x < (ORIGINAL_X0 + 302 - 10) &&
						TouchPoint.y > ORIGINAL_Y0 + 10 && TouchPoint.y < (ORIGINAL_Y0 + 402 - 10))  /* In range */
					{
						if(1 == gThickProf.FunOption.Is100_300)
						{
							DrawMan.currentPoint = 551 - TouchPoint.y;
							if(DrawMan.currentPoint > 399)DrawMan.currentPoint = 399;
						}
						else
						{
							DrawMan.currentPoint = (551 - TouchPoint.y + 1)/4 * 4;
							if(DrawMan.currentPoint > 396)DrawMan.currentPoint = 396;
						}
						DrawMan.step = S$STEP_ADDLINE;
						setColor = 2;
					}
				}
			}
			else
			{
				cntPressed = 0;
			}

			R_TRIG_DEL.CLK = delButton;
			R_TRIG(&R_TRIG_DEL);
			if(R_TRIG_DEL.Q == 1)
			{
				DrawMan.step = S$STEP_DELLINE;
			}

			R_TRIG_CURTOL.CLK = curtolButton;
			R_TRIG(&R_TRIG_CURTOL);
			if ( R_TRIG_CURTOL.Q ==1)
			{
				DrawMan.step = S$STEP_CURVETOL;
			}

			R_TRIG_Change.CLK = changeButton;
			R_TRIG(&R_TRIG_Change);
			if ( R_TRIG_Change.Q ==1)
			{
				bCurveIndexChgBtn = 1;
			}

			if(bCurveIndexChange == 1)
			{
				bCurveIndexChange = 0;
				bBackEnable = 0;
				bRedoEnable = 0;
				ChangeEnable = 1;
			}

			R_TRIG_CLEAR.CLK = clearButton;
			R_TRIG(&R_TRIG_CLEAR);
			if ( R_TRIG_CLEAR.Q ==1)
			{
				bBackEnable = 1;
				memcpy(&mDrawMan,&DrawMan,sizeof(mDrawMan));
				memcpy(&mCurveNode,&CurveNode,sizeof(mCurveNode));
				memcpy(&mSetPos,&SetPos,sizeof(mSetPos));

				DrawMan.step = S$STEP_CLAER;
			}
			break;

		case S$STEP_ADDLINE:
				moveInputEnable = 0;

			if (1 == upButton  || 1 == focusUpButton)
			{
			movePoint = 1;
			}
			else if (1 == downButton || 1 == focusDownButton)
			{
			movePoint = -1;
			}
			else
			{
			movePoint = 0;
			}

			/*move the cross cursor*/
			moveCross(&movePoint);

			if(1 == bAddLineMode)
			{
				if(1 == gThickProf.FunOption.Is100_300)
				{
					DrawMan.currentPoint = IndexAddLine * 4;
				}
				else
				{
					DrawMan.currentPoint = IndexAddLine;
				}
				setColor = 2;
				bAddLineMode = 0;
				IndexAddLine = 0;
			}

			if(0 == gPanelObj.vcHandle)
			{
				gPanelObj.vcHandle = VA_Setup(1, gPanelObj.VisualName);
			}

			if (gPanelObj.vcHandle != 0)
			{
				if (!VA_Saccess(1, gPanelObj.vcHandle))
				{
					VA_GetTouchAction (1,gPanelObj.vcHandle,0,(UDINT)(&TouchPoint));
					VA_Srelease(1, gPanelObj.vcHandle);
				}
			}

			if(1 == TouchPoint.status)
			{
				cntPressed = cntPressed + 1;

				if(10 == cntPressed)
				{
					if(TouchPoint.x > ORIGINAL_X0 + 10 && TouchPoint.x < (ORIGINAL_X0 + 302 - 10) &&
						TouchPoint.y > ORIGINAL_Y0 + 10 && TouchPoint.y < (ORIGINAL_Y0 + 402 - 10))  /* In range */
					{
						if(1 == gThickProf.FunOption.Is100_300)
						{
							DrawMan.currentPoint = 551 - TouchPoint.y;
							if(DrawMan.currentPoint > 399)DrawMan.currentPoint = 399;
						}
						else
						{
							DrawMan.currentPoint = (551 - TouchPoint.y + 1)/4 * 4;
							if(DrawMan.currentPoint > 396)DrawMan.currentPoint = 396;
						}
					}
					setColor = 2;
				}
			}
			else
			{
				cntPressed = 0;
			}

			/*add a vertical line*/
			R_TRIG_ENTER.CLK = tabButton;
			R_TRIG(&R_TRIG_ENTER);

			if ( R_TRIG_ENTER.Q ==1)
			{
				bBackEnable = 1;
				memcpy(&mDrawMan,&DrawMan,sizeof(mDrawMan));
				memcpy(&mCurveNode,&CurveNode,sizeof(mCurveNode));
				memcpy(&mSetPos,&SetPos,sizeof(mSetPos));

				addNode  = 1;
				nodeAdd(&addNode,DrawMan.currentPoint);
				DrawMan.currentNode 	= DrawMan.currentPoint;
				DrawMan.step = S$STEP_EDIT;
				DrawMan.flagLineFocus 	= 0;
				scanNode = 1;
			}

			/*esc the cross cursor*/
			F_TRIG_TAB.CLK = escButton;
			F_TRIG(&F_TRIG_TAB);
			if ( F_TRIG_TAB.Q ==1)
			{
				addNode 	  = 0;
				scanNode 	  = 1;
				DrawMan.step = S$STEP_EDIT;
			}

			tempIndex = DrawMan.currentPoint;
			break;

		case S$STEP_DELLINE:
			moveInputEnable = 0;

			if (DrawMan.flagLineFocus == 1 )
			{
				bBackEnable = 1;
				memcpy(&mDrawMan,&DrawMan,sizeof(mDrawMan));
				memcpy(&mCurveNode,&CurveNode,sizeof(mCurveNode));
				memcpy(&mSetPos,&SetPos,sizeof(mSetPos));

				delNode = 1;
				nodeDel(&delNode,DrawMan.currentNode);
			}
			DrawMan.step = S$STEP_EDIT;
			break;

		case S$STEP_CURVETOL:
			moveInputEnable = 0;

			if(DrawMan.flagLineFocus == 0)
			{
				bBackEnable = 1;
				memcpy(&mDrawMan,&DrawMan,sizeof(mDrawMan));
				memcpy(&mCurveNode,&CurveNode,sizeof(mCurveNode));
				memcpy(&mSetPos,&SetPos,sizeof(mSetPos));

				curveToL = 1;
				curveToLine((USINT *)(&curveToL),DrawMan.currentNode);
			}
			DrawMan.step = S$STEP_EDIT;
			break;

		case S$STEP_CURVEMOVE:
			moveInputEnable = 0;

			curveMove();
			moveValue = 0;
			DrawMan.step = S$STEP_EDIT;
			break;

		case S$STEP_UNDO:
			bRedoEnable = 1;
			memcpy(&redoDrawMan,&DrawMan,sizeof(DrawMan));
			memcpy(&redoCurveNode,&CurveNode,sizeof(CurveNode));
			memcpy(&redoSetPos,&SetPos,sizeof(SetPos));

			bBackEnable = 0;
			memcpy(&DrawMan,&mDrawMan,sizeof(mDrawMan));
			memcpy(&CurveNode,&mCurveNode,sizeof(mCurveNode));
			memcpy(&SetPos,&mSetPos,sizeof(mSetPos));

			DrawMan.draw = 1;
			DrawMan.step = S$STEP_EDIT;
			break;

		case S$STEP_REDO:
			bBackEnable = 1;
			memcpy(&mDrawMan,&DrawMan,sizeof(DrawMan));
			memcpy(&mCurveNode,&CurveNode,sizeof(CurveNode));
			memcpy(&mSetPos,&SetPos,sizeof(SetPos));

			bRedoEnable = 0;
			memcpy(&DrawMan,&redoDrawMan,sizeof(redoDrawMan));
			memcpy(&CurveNode,&redoCurveNode,sizeof(redoCurveNode));
			memcpy(&SetPos,&redoSetPos,sizeof(redoSetPos));

			DrawMan.draw = 1;
			DrawMan.step = S$STEP_EDIT;
			break;

		case S$STEP_CLAER:
			curveClear();
			DrawMan.draw = 1;
			DrawMan.step = S$STEP_EDIT;
			break;
	}/* switch (DrawMan.step) */

	if(DrawMan.step != S$STEP_ADDLINE)
	{
		bHideCrossImply = 1;
	}
	else
	{
		bHideCrossImply = 0;
	}

	if(DrawMan.step != S$STEP_EDIT || gPanelObj.PasswordLevel < 1)
	{
		bHideInsert       = 1;
		bHideCurveOperate = 1;
		bHideDel          = 1;
	}
	else
	{
		if(DrawMan.flagLineFocus == 1)
		{
			bHideInsert       = 0;
			bHideCurveOperate = 1;
			if(tempIndex != 0 && tempIndex != S$THICK_MAX)
			{
				bHideDel = 0;
			}
			else
			{
				bHideDel = 1;
			}
		}
		else
		{
			bHideInsert       = 0;
			bHideCurveOperate = 0;
			bHideDel          = 1;
		}
	}

	curveScan(&scanNode);
	curveQuickScan(&scanLine);
	curveColor(&setColor);
	weightSet();

	for(i=0;i<10;i++)
	{
		inputLock[i] = 0;
	}
	if(DrawMan.input > 9)DrawMan.input= 9;

	inputLock[DrawMan.input] = 1;

	cntFlash ++;
	if(cntFlash >= 10000)cntFlash = 0;

	if(0 != isDownLoad)
	{
		if((cntFlash % ((UINT)(1.0/tTask))) < (0.51/tTask))
		{
			loadBmpGrpFlash = 0;
		}
		else
		{
			loadBmpGrpFlash = 1;
		}
	}
	else
	{
		loadBmpGrpFlash = 0;
	}

}/*end of CYCLIC*/
/**************************************************************************************
**        				FUNCTION  REALIZE				   							 **
**************************************************************************************/
void nodeAdd(USINT *enable, UINT nodeNum)
{
	curveNode_typ    *p0,*p1;
	unsigned short   i;
	float			  t;

	if (*enable == 1) *enable = 0;
	else return;

	if (CurveNode[nodeNum].flagNode == 1 || nodeNum > S$THICK_MAX - 3 || nodeNum < 3)
	{
		strcpy(DrawMan.status,"can not add new node");
		return;
	}
	else
	{
		strcpy(DrawMan.status,"the new node is added");
		CurveNode[nodeNum].flagNode = 1;
	}

	for (i = 0 ; i<= S$THICK_MAX; i ++)
	{
		if ( CurveNode[i].next != 0 && CurveNode[i].next > nodeNum )
		{

			p0 = &CurveNode[nodeNum];
			p1 = &CurveNode[CurveNode[i].next];

			t	=(float)(SetPos[nodeNum].y - p1->v0.y)/(float)(p1->v3.y - p1->v0.y);

			p0->former   = i;
			p0->next     = CurveNode[i].next;

			CurveNode[i].next = nodeNum;

			p0->v0.x     = CurveNode[i].v3.x;
			p0->v0.y     = CurveNode[i].v3.y;

			p0->v1.x     = (1-t)*p1->v0.x + t*p1->v1.x;
			p0->v1.y     = (1-t)*p1->v0.y + t*p1->v1.y;
			p0->v2.x     = (1-t)*(1-t)*p1->v0.x + t*t*p1->v2.x + 2*t*(1-t)*p1->v1.x + 1;
			p0->v2.y     = (1-t)*(1-t)*p1->v0.y + t*t*p1->v2.y + 2*t*(1-t)*p1->v1.y;
			p0->v3.x     = SetPos[nodeNum].x;
			p0->v3.y     = SetPos[nodeNum].y;

			p1->v0.x     = p0->v3.x;
			p1->v0.y     = p0->v3.y;
			p1->v1.x     = (1-t)*(1-t)*p1->v1.x + 2*t*(1-t)*p1->v2.x + t*t*p1->v3.x + 1;
			p1->v1.y     = (1-t)*(1-t)*p1->v1.y + 2*t*(1-t)*p1->v2.y + t*t*p1->v3.y;
			p1->v2.x     = (1-t)*p1->v2.x + t*p1->v3.x + 1;
			p1->v2.y     = (1-t)*p1->v2.y + t*p1->v3.y;
			p1->v3.x     = p1->v3.x;
			p1->v3.y     = p1->v3.y;

			p1->former   = nodeNum;
			p0 = 0;
			p1 = 0;
			break;
		}
	}
} /*end of function*/

void nodeDel(USINT *enable,UINT nodeNum)
{
	UINT	oldNodeNum;
	*enable 	= 0;

	if (CurveNode[nodeNum].flagNode == 0 || nodeNum == 0 || nodeNum == S$THICK_MAX)
	{
		strcpy(DrawMan.status,"can not delete the node");
		return;
	}
	else
	{
		strcpy(DrawMan.status,"the node is deleted");
		CurveNode[nodeNum].flagNode = 0;
	}
	oldNodeNum  = CurveNode[nodeNum].next;
	CurveNode[CurveNode[nodeNum].former].next 	= CurveNode[nodeNum].next;
	CurveNode[oldNodeNum].former = CurveNode[nodeNum].former;
	CurveNode[oldNodeNum].v0.x   = CurveNode[nodeNum].v0.x;
	CurveNode[oldNodeNum].v0.y   = CurveNode[nodeNum].v0.y;
	CurveNode[oldNodeNum].v1.x   = CurveNode[nodeNum].v1.x;
	CurveNode[oldNodeNum].v1.y   = CurveNode[oldNodeNum].v0.y +
		(CurveNode[oldNodeNum].v3.y - CurveNode[oldNodeNum].v0.y)*1/
		S$THICK_V_SCALE;
	CurveNode[oldNodeNum].v2.y   = CurveNode[oldNodeNum].v0.y +
		(CurveNode[oldNodeNum].v3.y - CurveNode[oldNodeNum].v0.y)*(S$THICK_V_SCALE - 1)/
		S$THICK_V_SCALE;
	CurveNode[nodeNum].v0.x    = 0;
	CurveNode[nodeNum].v0.y    = 0;
	CurveNode[nodeNum].v1.x    = 0;
	CurveNode[nodeNum].v1.y    = 0;
	CurveNode[nodeNum].v2.x    = 0;
	CurveNode[nodeNum].v2.y    = 0;
	CurveNode[nodeNum].v3.x    = 0;
	CurveNode[nodeNum].v3.y    = 0;
	CurveNode[nodeNum].former  = 0;
	CurveNode[nodeNum].next    = 0;
	DrawMan.currentNode		  	 = oldNodeNum;

	DrawMan.flagLineFocus 	= 1;
	scanNode = -1;

}/*end of function*/

void curveScan(SINT *upDown)
{
	if (*upDown == 1)
	{
		if (DrawMan.flagLineFocus == 1)
		{
			if (DrawMan.currentNode != S$THICK_MAX)
				{
				DrawMan.flagLineFocus = 0;
				DrawMan.currentNode   = CurveNode[DrawMan.currentNode].next;
				DrawMan.v1 = CurveNode[DrawMan.currentNode].v1.x;
				DrawMan.v2 = CurveNode[DrawMan.currentNode].v2.x;
			}
			else
			{
				DrawMan.currentNode = 0;
				DrawMan.v2  = CurveNode[DrawMan.currentNode].v2.x;
				DrawMan.v03 = CurveNode[DrawMan.currentNode].v3.x;
				DrawMan.v1  = CurveNode[CurveNode[DrawMan.currentNode].next].v1.x;
			}
		}
		else
		{
			DrawMan.flagLineFocus = 1;
			DrawMan.v2   = CurveNode[DrawMan.currentNode].v2.x;
			DrawMan.v03  = CurveNode[DrawMan.currentNode].v3.x;
			DrawMan.v1   = CurveNode[CurveNode[DrawMan.currentNode].next].v1.x;
		}

		setColor = 1;
		*upDown = 0;
	}

	if(*upDown == -1)
	{
		if (DrawMan.flagLineFocus == 1)
		{
			if (DrawMan.currentNode != 0)
			{
				DrawMan.flagLineFocus = 0;
				DrawMan.v1 = CurveNode[DrawMan.currentNode].v1.x;
				DrawMan.v2 = CurveNode[DrawMan.currentNode].v2.x;
			}
			else
			{
				DrawMan.currentNode = S$THICK_MAX;
				DrawMan.v2   = CurveNode[DrawMan.currentNode].v2.x;
				DrawMan.v03  = CurveNode[DrawMan.currentNode].v3.x;
			}
		}
		else
		{
			DrawMan.flagLineFocus = 1;
			DrawMan.currentNode   = CurveNode[DrawMan.currentNode].former;
			DrawMan.v2	 = CurveNode[DrawMan.currentNode].v2.x;
			DrawMan.v03  = CurveNode[DrawMan.currentNode].v3.x;
			DrawMan.v1   = CurveNode[CurveNode[DrawMan.currentNode].next].v1.x;
		}
		setColor = 1;
		*upDown = 0;
	}

	strcpy(DrawMan.status,"scan finished");
}/*end of function*/

void curveQuickScan(SINT *upDown)
{
	if (*upDown == 1)
	{
		if (DrawMan.flagLineFocus == 1)
		{
			if (DrawMan.currentNode != S$THICK_MAX)
				{
				bStartUpLineFocus = 1;
				DrawMan.flagLineFocus = 0;
				DrawMan.currentNode   = CurveNode[DrawMan.currentNode].next;
				DrawMan.v1	= CurveNode[DrawMan.currentNode].v1.x;
				DrawMan.v2  = CurveNode[DrawMan.currentNode].v2.x;
			}
			else
			{
				bStartUpLineFocus   = 0;
				DrawMan.currentNode = 0;
				DrawMan.v2   = CurveNode[DrawMan.currentNode].v2.x;
				DrawMan.v03  = CurveNode[DrawMan.currentNode].v3.x;
				DrawMan.v1   = CurveNode[CurveNode[DrawMan.currentNode].next].v1.x;
			}
		}
		else
		{
			bStartUpLineFocus     = 0;
			DrawMan.flagLineFocus = 1;
			DrawMan.v2   = CurveNode[DrawMan.currentNode].v2.x;
			DrawMan.v03  = CurveNode[DrawMan.currentNode].v3.x;
			DrawMan.v1   = CurveNode[CurveNode[DrawMan.currentNode].next].v1.x;
		}

		if(1 == bStartUpLineFocus)
		{
			if (DrawMan.flagLineFocus == 1)
			{
				if (DrawMan.currentNode != S$THICK_MAX)
					{
					DrawMan.flagLineFocus = 0;
					DrawMan.currentNode   = CurveNode[DrawMan.currentNode].next;
					DrawMan.v1	= CurveNode[DrawMan.currentNode].v1.x;
					DrawMan.v2  = CurveNode[DrawMan.currentNode].v2.x;
				}
				else
				{
					DrawMan.currentNode = 0;
					DrawMan.v2   = CurveNode[DrawMan.currentNode].v2.x;
					DrawMan.v03  = CurveNode[DrawMan.currentNode].v3.x;
					DrawMan.v1   = CurveNode[CurveNode[DrawMan.currentNode].next].v1.x;
				}
			}
			else
			{
				DrawMan.flagLineFocus = 1;
				DrawMan.v2   = CurveNode[DrawMan.currentNode].v2.x;
				DrawMan.v03  = CurveNode[DrawMan.currentNode].v3.x;
				DrawMan.v1   = CurveNode[CurveNode[DrawMan.currentNode].next].v1.x;
			}
		}

		setColor = 1;
		*upDown = 0;
	}

	if(*upDown == -1)
	{
		if (DrawMan.flagLineFocus == 1)
		{
			if (DrawMan.currentNode != 0)
			{
				bStartDnLineFocus     = 1;
				DrawMan.flagLineFocus = 0;
				DrawMan.v1 = CurveNode[DrawMan.currentNode].v1.x;
				DrawMan.v2 = CurveNode[DrawMan.currentNode].v2.x;
			}
			else
			{
				bStartDnLineFocus   = 0;
				DrawMan.currentNode = S$THICK_MAX;
				DrawMan.v2  = CurveNode[DrawMan.currentNode].v2.x;
				DrawMan.v03 = CurveNode[DrawMan.currentNode].v3.x;
			}
		}
		else
		{
			bStartDnLineFocus     = 0;
			DrawMan.flagLineFocus = 1;
			DrawMan.currentNode   = CurveNode[DrawMan.currentNode].former;
			DrawMan.v2	= CurveNode[DrawMan.currentNode].v2.x;
			DrawMan.v03 = CurveNode[DrawMan.currentNode].v3.x;
			DrawMan.v1  = CurveNode[CurveNode[DrawMan.currentNode].next].v1.x;
		}

		if(1 == bStartDnLineFocus)
		{
			if (DrawMan.flagLineFocus == 1)
			{
				if (DrawMan.currentNode != 0)
				{
					DrawMan.flagLineFocus = 0;
					DrawMan.v1 = CurveNode[DrawMan.currentNode].v1.x;
					DrawMan.v2 = CurveNode[DrawMan.currentNode].v2.x;
				}
				else
				{
					DrawMan.currentNode = S$THICK_MAX;
					DrawMan.v2  = CurveNode[DrawMan.currentNode].v2.x;
					DrawMan.v03 = CurveNode[DrawMan.currentNode].v3.x;
				}
			}
			else
			{
				DrawMan.flagLineFocus = 1;
				DrawMan.currentNode   = CurveNode[DrawMan.currentNode].former;
				DrawMan.v2	= CurveNode[DrawMan.currentNode].v2.x;
				DrawMan.v03 = CurveNode[DrawMan.currentNode].v3.x;
				DrawMan.v1  = CurveNode[CurveNode[DrawMan.currentNode].next].v1.x;
			}
		}

		setColor = 1;
		*upDown  = 0;
	}

	strcpy(DrawMan.status,"quick scan finished");
}/*end of function*/

void vxEdit()
{
	if (DrawMan.flagLineFocus == 0)
	{
		if ( v1Add == 1)
		{
			counter0++;
			counter1++;
			if (counter1 == 1) DrawMan.v1 = DrawMan.v1 + 3;
			else if (counter1 < 4);
			else if (counter1 < 8) DrawMan.v1 = DrawMan.v1 + StepLength/2;
			else DrawMan.v1 = DrawMan.v1 + StepLength;
		}
		else if ( v1Sub == 1)
		{
			counter0++;
			counter1++;
			if (counter1 == 1) DrawMan.v1 = DrawMan.v1 - 3;
			else if (counter1 < 4);
			else if (counter1 < 8) DrawMan.v1 =DrawMan.v1 - StepLength/2;
			else DrawMan.v1 =DrawMan.v1  - StepLength;
		}
		else if ( v2Add == 1)
		{
			counter0++;
			counter1++;
			if (counter1 == 1) DrawMan.v2 = DrawMan.v2 + 3;
			else if (counter1 < 4);
			else if (counter1 < 8)DrawMan.v2 = DrawMan.v2 + StepLength/2;
			else DrawMan.v2 = DrawMan.v2 + StepLength;
		}
		else if ( v2Sub == 1)
		{
			counter0++;
			counter1++;
			if (counter1 == 1) DrawMan.v2 = DrawMan.v2 - 3;
			else if (counter1 < 4);
			else if (counter1 < 8)DrawMan.v2 = DrawMan.v2 - StepLength/2;
			else DrawMan.v2 = DrawMan.v2 - StepLength;
		}
		else
		{
			counter0 = 0;
			counter1 = 0;
		}
	}
	else
	{
		tempGap = currentGap - oldcurrentGap;

		if (inputok == 1)
		{
			bBackEnable = 1;
			memcpy(&mDrawMan,&DrawMan,sizeof(mDrawMan));
			memcpy(&mCurveNode,&CurveNode,sizeof(mCurveNode));
			memcpy(&mSetPos,&SetPos,sizeof(mSetPos));

			DrawMan.v1 = DrawMan.v1 + tempGap;
			DrawMan.v2 = DrawMan.v2 + tempGap;
			DrawMan.v03 = currentGap;
			inputok = 0;
		}

		if ( v03Sub == 1)
		{
			counter0++;
			counter1++;
			if (counter1 == 1)
			{
				if (DrawMan.v03 > (DrawMan.weight))
				{
					DrawMan.v1  = DrawMan.v1  - 3;
					DrawMan.v2  = DrawMan.v2  - 3;
					DrawMan.v03 = DrawMan.v03 - 3;
				}
			}
			else if (counter1 < 4);
			else if (counter1 < 8)
			{
				if (DrawMan.v03 > (DrawMan.weight))
				{
					DrawMan.v1  = DrawMan.v1  - StepLength/2;
					DrawMan.v2  = DrawMan.v2  - StepLength/2;
					DrawMan.v03 = DrawMan.v03 - StepLength/2;
				}
			}
			else
			{
				if (DrawMan.v03 > (DrawMan.weight))
				{
					DrawMan.v1 = DrawMan.v1  - StepLength;
					DrawMan.v2 = DrawMan.v2  - StepLength;
					DrawMan.v03= DrawMan.v03 - StepLength;
				}
			}
		}
		else if ( v03Add == 1)
		{
			counter0++;
			counter1++;

			if (counter1 == 1)
			{
				if (DrawMan.v03 < 2970)
				{
					DrawMan.v1  = DrawMan.v1  + 3;
					DrawMan.v2  = DrawMan.v2  + 3;
					DrawMan.v03 = DrawMan.v03 + 3;
				}
			}
			else if (counter1 < 4);
			else if (counter1 < 8)
			{
				if (DrawMan.v03 < 2970)
				{
					DrawMan.v1  = DrawMan.v1  + StepLength/2;
					DrawMan.v2  = DrawMan.v2  + StepLength/2;
					DrawMan.v03 = DrawMan.v03 + StepLength/2;
				}
			}
			else
			{
				if (DrawMan.v03 < 2970)
				{
					DrawMan.v1 = DrawMan.v1  + StepLength;
					DrawMan.v2 = DrawMan.v2  + StepLength;
					DrawMan.v03= DrawMan.v03 + StepLength;
				}
			}
		}
		else
		{
			counter0 = 0;
			counter1 = 0;
		}
	}
}/*end of function*/

void vxEditUnit(INT unitLength)
{
	if(unitLength < 0)unitLength = -unitLength;
	if(unitLength < 3)unitLength = 3;

	if (DrawMan.flagLineFocus == 0)
	{
		if ( v1Add == 1)
		{
			counter0++;
			counter1++;
			if (counter1 == 1) DrawMan.v1 = DrawMan.v1 + 3;
			else if (counter1 < 4);
			else if (counter1 < 8) DrawMan.v1 = DrawMan.v1 + StepLength/2;
			else DrawMan.v1 = DrawMan.v1 + StepLength;
		}
		else if ( v1Sub == 1)
		{
			counter0++;
			counter1++;
			if (counter1 == 1) DrawMan.v1 = DrawMan.v1 - 3;
			else if (counter1 < 4);
			else if (counter1 < 8) DrawMan.v1 =DrawMan.v1 - StepLength/2;
			else DrawMan.v1 =DrawMan.v1  - StepLength/2;
		}
		else if ( v2Add == 1)
		{
			counter0++;
			counter1++;
			if (counter1 == 1) DrawMan.v2 = DrawMan.v2 + 3;
			else if (counter1 < 4);
			else if (counter1 < 8)DrawMan.v2 = DrawMan.v2 + StepLength/2;
			else DrawMan.v2 = DrawMan.v2 + StepLength;
		}
		else if ( v2Sub == 1)
		{
			counter0++;
			counter1++;
			if (counter1 == 1) DrawMan.v2 = DrawMan.v2 - 3;
			else if (counter1 < 4);
			else if (counter1 < 8)DrawMan.v2 = DrawMan.v2 - StepLength/2;
			else DrawMan.v2 = DrawMan.v2 - StepLength;
		}
		else
		{
			counter0 = 0;
			counter1 = 0;
		}
	}
	else
	{
		if(currentGap < DrawMan.weight + 30)currentGap = DrawMan.weight + 30;
		tempGap = ((INT)currentGap) - oldcurrentGap;

		if (inputok == 1)
		{
			bBackEnable = 1;
			memcpy(&mDrawMan,&DrawMan,sizeof(mDrawMan));
			memcpy(&mCurveNode,&CurveNode,sizeof(mCurveNode));
			memcpy(&mSetPos,&SetPos,sizeof(mSetPos));

			DrawMan.v1 = DrawMan.v1 + tempGap;
			DrawMan.v2 = DrawMan.v2 + tempGap;
			DrawMan.v03 = currentGap;
			inputok = 0;
		}

		if ( v03Sub == 1)
		{
			counter0++;
			counter1++;
			if (counter1 == 1)
			{
				if (DrawMan.v03 > (DrawMan.weight + unitLength))
				{
					DrawMan.v1  = DrawMan.v1  - unitLength;
					DrawMan.v2  = DrawMan.v2  - unitLength;
					DrawMan.v03 = DrawMan.v03 - unitLength;
				}
			}
			else if (counter1 < 4);
			else if ((counter1 % 2) == 0)
			{
				if (DrawMan.v03 > (DrawMan.weight + unitLength))
				{
					DrawMan.v1  = DrawMan.v1  - unitLength;
					DrawMan.v2  = DrawMan.v2  - unitLength;
					DrawMan.v03 = DrawMan.v03 - unitLength;
				}
			}
			else;
		}
		else if ( v03Add == 1)
		{
			counter0++;
			counter1++;

			if (counter1 == 1)
			{
				if (DrawMan.v03 < 2970 - unitLength)
				{
					DrawMan.v1  = DrawMan.v1  + unitLength;
					DrawMan.v2  = DrawMan.v2  + unitLength;
					DrawMan.v03 = DrawMan.v03 + unitLength;
				}
			}
			else if (counter1 < 4);
			else if ((counter1 % 2) == 0)
			{
				if (DrawMan.v03 < 2970 - unitLength)
				{
					DrawMan.v1  = DrawMan.v1  + unitLength;
					DrawMan.v2  = DrawMan.v2  + unitLength;
					DrawMan.v03 = DrawMan.v03 + unitLength;
				}
			}
			else;
		}
		else
		{
			counter0 = 0;
			counter1 = 0;
		}
	}
}/*end of function*/

void moveCross(SINT *upDown)
{
	if(0 == gThickProf.FunOption.Is100_300)
	{
		nodeIdxInc = 1;
	}
	else
	{
		nodeIdxInc = 4;
	}

	if (*upDown == 1)
	{
		counter0++;
		counter1++;

		if (counter1 == 1)DrawMan.currentPoint = DrawMan.currentPoint + nodeIdxInc;
		else if (counter1 < 10);
		else
		{
			DrawMan.currentPoint = DrawMan.currentPoint + nodeIdxInc;
		}

		if (DrawMan.currentPoint > S$THICK_MAX) DrawMan.currentPoint = 0;

		if(1 == gThickProf.FunOption.Is100_300)
		{
			DrawMan.currentPoint = DrawMan.currentPoint/4 * 4;
		}

	}
	else if (*upDown == -1)
	{
		counter0++;
		counter1++;

		if (counter1 == 1) DrawMan.currentPoint = DrawMan.currentPoint - nodeIdxInc;
		else if (counter1 < 10);
		else
		{
			DrawMan.currentPoint = DrawMan.currentPoint - nodeIdxInc;
		}

		if (DrawMan.currentPoint < 0) DrawMan.currentPoint = S$THICK_MAX ;

		if(1 == gThickProf.FunOption.Is100_300)
		{
			DrawMan.currentPoint = DrawMan.currentPoint/4 * 4;
		}
	}
	else
	{
		counter0 = 0;
		counter1 = 0;
	}

	if (*upDown != 0) DrawMan.draw = 1;

}/*end of function*/

void curveColor(USINT *action)
{
	if (*action == 0) return;
	if (*action != 0)
	{
		for (i = 0 ; i <= S$THICK_MAX; i ++)
			{
			CurveNode[i].color 		= unfocusColor;
			CurveNode[i].vLineColor = unfocusColor;
		}
	}

	if (*action == 1)
	{
		if (DrawMan.flagLineFocus == 1)
		{
			CurveNode[DrawMan.currentNode].vLineColor = focusColor;
		}
		else
		{
			for(i=CurveNode[DrawMan.currentNode].former;i<=DrawMan.currentNode;i++)
			{
				CurveNode[i].color = focusColor;
			}
		}
	}

	*action 	= 0;
	DrawMan.draw = 1;
}/*end of function*/

void weightSet()
{
	switch (weightStep)
	{
		case 0:
			if(LengthUnit < 3)LengthUnit =3;
			if(LengthUnit > 150)LengthUnit = 150;
			if(1 == weightUpButton)
			{
				cntTime0++;

				if(cntTime0 == 1)
				{
					if(0 == gThickProf.FunOption.bLengthUnit)
					{
						DrawMan.weight = DrawMan.weight + 3;
					}
					else
					{
						DrawMan.weight = DrawMan.weight + LengthUnit;
					}
				}
			}
			else if (1 == weightDownButton)
			{
				cntTime0++;

				if(cntTime0 == 1)
				{
					if(0 == gThickProf.FunOption.bLengthUnit)
					{
						DrawMan.weight = DrawMan.weight - 3;
					}
					else
					{
						DrawMan.weight = DrawMan.weight - LengthUnit;
					}
				}
			}
			else
			{
				cntTime0 = 0;
			}

			if (DrawMan.oldWeight != DrawMan.weight)
			{
				if( DrawMan.oldWeight >=0 && DrawMan.weight >= 0)
				{
					bBackEnable = 1;
					memcpy(&mDrawMan,&DrawMan,sizeof(mDrawMan));
					mDrawMan.weight = mDrawMan.oldWeight;
					memcpy(&mCurveNode,&CurveNode,sizeof(mCurveNode));
					memcpy(&mSetPos,&SetPos,sizeof(mSetPos));

					weightStep = 10;			/* positive vlaue */
				}
				else if( DrawMan.oldWeight >= 0 && DrawMan.weight < 0)
				{
					bBackEnable = 1;
					memcpy(&mDrawMan,&DrawMan,sizeof(mDrawMan));
					mDrawMan.weight = mDrawMan.oldWeight;
					memcpy(&mCurveNode,&CurveNode,sizeof(mCurveNode));
					memcpy(&mSetPos,&SetPos,sizeof(mSetPos));

					weightStep = 110; 		/* negative negative vlaue */
				}
				else
				{
					DrawMan.weight = DrawMan.oldWeight;
					weightStep = 0;
				}
			}
			break;

		/* positive weight  */
		case 10:
			for (i = 0 ; i<= S$THICK_MAX; i ++)
				{
				if ((SetPos[i].x + (DrawMan.weight - DrawMan.oldWeight)) > S$THICK_X_LENGTH ||
						(SetPos[i].x + (DrawMan.weight - DrawMan.oldWeight)) < 3)    //6//ipis0619
					{
					DrawMan.weight = DrawMan.oldWeight;
					weightStep = 0;
					break;
				}
				else if (i == S$THICK_MAX) weightStep = 20;
			}
			break;
		case 20:
			for (i = 0 ; i<= S$THICK_MAX; i ++)
				{
				SetPos[i].x += ((DrawMan.weight - DrawMan.oldWeight));
				if (CurveNode[i].flagNode == 1)
				{
					CurveNode[i].v0.x += ((DrawMan.weight - DrawMan.oldWeight));
					CurveNode[i].v1.x += ((DrawMan.weight - DrawMan.oldWeight));
					CurveNode[i].v2.x += ((DrawMan.weight - DrawMan.oldWeight));
					CurveNode[i].v3.x += ((DrawMan.weight - DrawMan.oldWeight));
				}
			}
			DrawMan.v1 	+= ((DrawMan.weight - DrawMan.oldWeight));
			DrawMan.v2 	+= ((DrawMan.weight - DrawMan.oldWeight));
			DrawMan.v03 += ((DrawMan.weight - DrawMan.oldWeight));
			DrawMan.oldWeight = DrawMan.weight =0; //ipis0619
			weightStep = 0;
			break;

		/* negative weight  */
		case 110:
			for (i = 0 ; i<= S$THICK_MAX; i ++)
				{
				if ((SetPos[i].x + (DrawMan.weight - DrawMan.oldWeight)) > S$THICK_X_LENGTH ||
						(SetPos[i].x + (DrawMan.weight - DrawMan.oldWeight)) < 6)
					{
					DrawMan.weight = DrawMan.oldWeight;
					weightStep = 0;
					break;
				}
				else if (i == S$THICK_MAX) weightStep = 120;
			}
			break;
		case 120:
			for (i = 0 ; i<= S$THICK_MAX; i ++)
				{
				SetPos[i].x += ((DrawMan.weight - DrawMan.oldWeight));
				if (CurveNode[i].flagNode == 1)
				{
					CurveNode[i].v0.x += ((DrawMan.weight - DrawMan.oldWeight));
					CurveNode[i].v1.x += ((DrawMan.weight - DrawMan.oldWeight));
					CurveNode[i].v2.x += ((DrawMan.weight - DrawMan.oldWeight));
					CurveNode[i].v3.x += ((DrawMan.weight - DrawMan.oldWeight));
				}
			}
			DrawMan.v1 	+= ((DrawMan.weight - DrawMan.oldWeight));
			DrawMan.v2 	+= ((DrawMan.weight - DrawMan.oldWeight));
			DrawMan.v03 += ((DrawMan.weight - DrawMan.oldWeight));
			DrawMan.oldWeight = DrawMan.weight = 0;
			weightStep = 0;
			break;
	}
}/*end of function*/

void curveToLine(USINT *action,UINT nodeNum)
{
	if (*action == 0) return;
	*action = 0;
	if (DrawMan.flagLineFocus == 0)
	{
		CurveNode[nodeNum].v1.x   	= 1 + CurveNode[nodeNum].v0.x +
			(CurveNode[nodeNum].v3.x - CurveNode[nodeNum].v0.x)*1/
			S$THICK_V_SCALE;
		CurveNode[nodeNum].v2.x   	= 1 + CurveNode[nodeNum].v0.x +
			(CurveNode[nodeNum].v3.x - CurveNode[nodeNum].v0.x)*(S$THICK_V_SCALE - 1)/
			S$THICK_V_SCALE;
	}
	DrawMan.flagLineFocus 	= 1;
	scanNode 				= -1;
}/*end of function*/

void curveMove()
{
	INT idx,idxMove;
	float t;

	memset(tempCurveNode,0,sizeof(tempCurveNode));

	if(moveValue > 20 || moveValue < -20)return;

	idxMove = 3 * moveValue;

	if(idxMove < 0)idxMove=-idxMove;

	if(moveValue > 0)
	{
		/* ------------ first node ------------ */
		tempCurveNode[0].former   = S$THICK_MAX;
		tempCurveNode[0].next     = idxMove;
		tempCurveNode[0].flagNode = 1;
		tempCurveNode[0].v3.x     = SetPos[0].x;

		/* ------------ second node ------------ */
		tempCurveNode[idxMove].former = 0;
		tempCurveNode[idxMove].next = CurveNode[0].next + idxMove;
		if(tempCurveNode[idxMove].next > S$THICK_MAX)tempCurveNode[idxMove].next = S$THICK_MAX;

		tempCurveNode[idxMove].flagNode = 1;

		tempCurveNode[idxMove].v0.x = SetPos[0].x;
		tempCurveNode[idxMove].v0.y = 0;

		tempCurveNode[idxMove].v1.x = SetPos[0].x+1;
		tempCurveNode[idxMove].v1.y = idxMove/3;

		tempCurveNode[idxMove].v2.x = SetPos[0].x+1;
		tempCurveNode[idxMove].v2.y = idxMove - idxMove/3;

		tempCurveNode[idxMove].v3.x = SetPos[0].x;
		tempCurveNode[idxMove].v3.y = idxMove;

		endIdx = 0;
		for (idx = 1; idx<= S$THICK_MAX -1; idx ++)
		{
			if(1 == CurveNode[idx].flagNode)
			{
				if(CurveNode[idx].next >= S$THICK_MAX - idxMove && idx < S$THICK_MAX - idxMove)
					{
					endIdx = idx;
					break;
				}
			}
		}

		for (idx = 1; idx< endIdx; idx ++)
		{
			if(1 == CurveNode[idx].flagNode)
			{
				tempCurveNode[idx + idxMove] = CurveNode[idx];

				tempCurveNode[idx + idxMove].former = CurveNode[idx].former + idxMove;
				tempCurveNode[idx + idxMove].next   = CurveNode[idx].next   + idxMove;
				if(tempCurveNode[idx + idxMove].next > S$THICK_MAX)tempCurveNode[idx + idxMove].next = S$THICK_MAX;

				tempCurveNode[idx + idxMove].v0.y = CurveNode[idx].v0.y + idxMove;
				tempCurveNode[idx + idxMove].v1.y = CurveNode[idx].v1.y + idxMove;
				tempCurveNode[idx + idxMove].v2.y = CurveNode[idx].v2.y + idxMove;
				tempCurveNode[idx + idxMove].v3.y = CurveNode[idx].v3.y + idxMove;
			}
		}

		if(CurveNode[S$THICK_MAX - idxMove].flagNode != 1)
		{
			if(endIdx != 0)
			{
				tempCurveNode[endIdx + idxMove] = CurveNode[endIdx];

				tempCurveNode[endIdx + idxMove].former = CurveNode[endIdx].former + idxMove;
				tempCurveNode[endIdx + idxMove].next   = S$THICK_MAX;

				tempCurveNode[endIdx + idxMove].v0.y = CurveNode[endIdx].v0.y + idxMove;
				tempCurveNode[endIdx + idxMove].v1.y = CurveNode[endIdx].v1.y + idxMove;
				tempCurveNode[endIdx + idxMove].v2.y = CurveNode[endIdx].v2.y + idxMove;
				tempCurveNode[endIdx + idxMove].v3.y = CurveNode[endIdx].v3.y + idxMove;
			}

			t =(float)(S$THICK_MAX - idxMove - CurveNode[CurveNode[endIdx].next].v0.y)/(float)(CurveNode[CurveNode[endIdx].next].v3.y -
				CurveNode[CurveNode[endIdx].next].v0.y);

				tempCurveNode[S$THICK_MAX].former = endIdx + idxMove;
			tempCurveNode[S$THICK_MAX].next   = 0;

			tempCurveNode[S$THICK_MAX].flagNode = 1;

			tempCurveNode[S$THICK_MAX].v0.x = CurveNode[CurveNode[endIdx].next].v0.x;
			tempCurveNode[S$THICK_MAX].v0.y = CurveNode[CurveNode[endIdx].next].v0.y + idxMove;

			tempCurveNode[S$THICK_MAX].v1.x = (1-t)*CurveNode[CurveNode[endIdx].next].v0.x + t*CurveNode[CurveNode[endIdx].next].v1.x;
			tempCurveNode[S$THICK_MAX].v1.y = (1-t)*CurveNode[CurveNode[endIdx].next].v0.y + t*CurveNode[CurveNode[endIdx].next].v1.y;
			tempCurveNode[S$THICK_MAX].v1.y = tempCurveNode[S$THICK_MAX].v1.y + idxMove;

			tempCurveNode[S$THICK_MAX].v2.x = (1-t)*(1-t)*CurveNode[CurveNode[endIdx].next].v0.x +
				t*t*CurveNode[CurveNode[endIdx].next].v2.x + 2*t*(1-t)*CurveNode[CurveNode[endIdx].next].v1.x;
			tempCurveNode[S$THICK_MAX].v2.y = (1-t)*(1-t)*CurveNode[CurveNode[endIdx].next].v0.y +
				t*t*CurveNode[CurveNode[endIdx].next].v2.y + 2*t*(1-t)*CurveNode[CurveNode[endIdx].next].v1.y;
			tempCurveNode[S$THICK_MAX].v2.y = tempCurveNode[S$THICK_MAX].v2.y + idxMove;

			tempCurveNode[S$THICK_MAX].v3.x = SetPos[S$THICK_MAX - idxMove].x;
			tempCurveNode[S$THICK_MAX].v3.y = S$THICK_MAX;
		}
		else
		{
			if(endIdx != 0)
			{
				tempCurveNode[endIdx + idxMove] = CurveNode[endIdx];

				tempCurveNode[endIdx + idxMove].former = CurveNode[endIdx].former + idxMove;
				tempCurveNode[endIdx + idxMove].next   = S$THICK_MAX;

				tempCurveNode[endIdx + idxMove].v0.y = CurveNode[endIdx].v0.y + idxMove;
				tempCurveNode[endIdx + idxMove].v1.y = CurveNode[endIdx].v1.y + idxMove;
				tempCurveNode[endIdx + idxMove].v2.y = CurveNode[endIdx].v2.y + idxMove;
				tempCurveNode[endIdx + idxMove].v3.y = CurveNode[endIdx].v3.y + idxMove;
			}

			tempCurveNode[S$THICK_MAX] = CurveNode[S$THICK_MAX - idxMove];

				tempCurveNode[S$THICK_MAX].former = endIdx + idxMove;
			tempCurveNode[S$THICK_MAX].next   = 0;

			tempCurveNode[S$THICK_MAX].v0.y = CurveNode[S$THICK_MAX - idxMove].v0.y + idxMove;
			tempCurveNode[S$THICK_MAX].v1.y = CurveNode[S$THICK_MAX - idxMove].v1.y + idxMove;
			tempCurveNode[S$THICK_MAX].v2.y = CurveNode[S$THICK_MAX - idxMove].v2.y + idxMove;
			tempCurveNode[S$THICK_MAX].v3.y = S$THICK_MAX;
		}

		memcpy(CurveNode,tempCurveNode,sizeof(CurveNode));

		for (idx = idxMove; idx<= S$THICK_MAX; idx ++)
		{
			tempSetPos[idx].x= SetPos[idx-idxMove].x;
			tempSetPos[idx].y = idx;
		}

		for (idx = 0; idx<idxMove; idx ++)
		{
			tempSetPos[idx].x = SetPos[0].x;
			tempSetPos[idx].y = idx;
		}

		memcpy(SetPos,tempSetPos,sizeof(SetPos));
	}
	else
	{
		startIdx = S$THICK_MAX;
		for (idx = S$THICK_MAX; idx > 1 ; idx --)
		{
			if(1 == CurveNode[idx].flagNode)
			{
				if(CurveNode[idx].v0.y < idxMove && idx <= CurveNode[idx].v3.y)
				{
					startIdx = idx;
					break;
				}
			}
		}

		if(CurveNode[idxMove].flagNode != 1)
		{
			tempCurveNode[0].former   = S$THICK_MAX;
			if(startIdx != 0)
			{
				tempCurveNode[0].next = startIdx - idxMove;
			}
			else
			{
				tempCurveNode[0].next = S$THICK_MAX - idxMove;
			}
			tempCurveNode[0].flagNode = 1;

			tempCurveNode[0].v3.x     = SetPos[idxMove].x;
			tempCurveNode[0].v3.y     = 0;

			tempCurveNode[tempCurveNode[0].next].former = 0;
			if(startIdx == S$THICK_MAX)
				{
				tempCurveNode[tempCurveNode[0].next].next = S$THICK_MAX;
			}
			else
			{
				tempCurveNode[tempCurveNode[0].next].next = CurveNode[startIdx].next - idxMove;
			}
			tempCurveNode[tempCurveNode[0].next].flagNode = 1;

			t =(float)(idxMove - CurveNode[startIdx].v0.y)/(float)(CurveNode[startIdx].v3.y - CurveNode[startIdx].v0.y);

			tempCurveNode[tempCurveNode[0].next].v0.x = SetPos[idxMove].x;
			tempCurveNode[tempCurveNode[0].next].v0.y = 0;

			tempCurveNode[tempCurveNode[0].next].v1.x = (1-t)*(1-t)*CurveNode[startIdx].v1.x + 2*t*(1-t)*CurveNode[startIdx].v2.x + t*t*CurveNode[startIdx].v3.x + 1;
			tempCurveNode[tempCurveNode[0].next].v1.y = (1-t)*(1-t)*CurveNode[startIdx].v1.y + 2*t*(1-t)*CurveNode[startIdx].v2.y + t*t*CurveNode[startIdx].v3.y;
			tempCurveNode[tempCurveNode[0].next].v1.y = tempCurveNode[tempCurveNode[0].next].v1.y - idxMove;

			tempCurveNode[tempCurveNode[0].next].v2.x = (1-t)*CurveNode[startIdx].v2.x + t*CurveNode[startIdx].v3.x + 1;
			tempCurveNode[tempCurveNode[0].next].v2.y = (1-t)*CurveNode[startIdx].v2.y + t*CurveNode[startIdx].v3.y;
			tempCurveNode[tempCurveNode[0].next].v2.y = tempCurveNode[tempCurveNode[0].next].v2.y - idxMove;

			tempCurveNode[tempCurveNode[0].next].v3.x = CurveNode[startIdx].v3.x;
			tempCurveNode[tempCurveNode[0].next].v3.y = CurveNode[startIdx].v3.y;
			tempCurveNode[tempCurveNode[0].next].v3.y = tempCurveNode[tempCurveNode[0].next].v3.y - idxMove;
		}
		else
		{
			tempCurveNode[0].former = S$THICK_MAX;
			tempCurveNode[0].next   = CurveNode[startIdx].next - idxMove;
			tempCurveNode[0].flagNode = 1;

			tempCurveNode[0].v3.x     = SetPos[idxMove].x;
			tempCurveNode[0].v3.y     = 0;
		}

		for (idx = startIdx + 1; idx< S$THICK_MAX; idx ++)
		{
			if(1 == CurveNode[idx].flagNode)
			{
				tempCurveNode[idx - idxMove] = CurveNode[idx];

				if(CurveNode[idx].former != 0)
				{
					tempCurveNode[idx - idxMove].former = CurveNode[idx].former - idxMove;
				}
				else
				{
					tempCurveNode[idx - idxMove].former = 0;
				}

				tempCurveNode[idx - idxMove].next = CurveNode[idx].next - idxMove;

				tempCurveNode[idx - idxMove].v0.y = CurveNode[idx].v0.y - idxMove;
				tempCurveNode[idx - idxMove].v1.y = CurveNode[idx].v1.y - idxMove;
				tempCurveNode[idx - idxMove].v2.y = CurveNode[idx].v2.y - idxMove;
				tempCurveNode[idx - idxMove].v3.y = CurveNode[idx].v3.y - idxMove;
			}
		}

		if(startIdx != S$THICK_MAX)
		{
			tempCurveNode[S$THICK_MAX - idxMove] = CurveNode[S$THICK_MAX];

				tempCurveNode[S$THICK_MAX - idxMove].former = CurveNode[S$THICK_MAX].former - idxMove;
			tempCurveNode[S$THICK_MAX - idxMove].next   = S$THICK_MAX;
			tempCurveNode[S$THICK_MAX - idxMove].flagNode = 1;

			tempCurveNode[S$THICK_MAX - idxMove].v0.y = CurveNode[idx].v0.y - idxMove;
			tempCurveNode[S$THICK_MAX - idxMove].v1.y = CurveNode[idx].v1.y - idxMove;
			tempCurveNode[S$THICK_MAX - idxMove].v2.y = CurveNode[idx].v2.y - idxMove;
			tempCurveNode[S$THICK_MAX - idxMove].v3.y = CurveNode[idx].v3.y - idxMove;
		}

		tempCurveNode[S$THICK_MAX].former = S$THICK_MAX - idxMove;
		tempCurveNode[S$THICK_MAX].next   = 0;
		tempCurveNode[S$THICK_MAX].flagNode = 1;

		tempCurveNode[S$THICK_MAX].v0.x = SetPos[S$THICK_MAX].x;
		tempCurveNode[S$THICK_MAX].v0.y = S$THICK_MAX - idxMove;

		tempCurveNode[S$THICK_MAX].v1.x = SetPos[S$THICK_MAX].x + 1;
		tempCurveNode[S$THICK_MAX].v1.y = S$THICK_MAX - idxMove * 2/3;

		tempCurveNode[S$THICK_MAX].v2.x = SetPos[S$THICK_MAX].x + 1;
		tempCurveNode[S$THICK_MAX].v2.y = S$THICK_MAX - idxMove/3;

		tempCurveNode[S$THICK_MAX].v3.x = SetPos[S$THICK_MAX].x;
		tempCurveNode[S$THICK_MAX].v3.y = S$THICK_MAX ;

		memcpy(CurveNode,tempCurveNode,sizeof(CurveNode));

		for (idx = S$THICK_MAX; idx> S$THICK_MAX -idxMove; idx --)
		{
			tempSetPos[idx].x = SetPos[S$THICK_MAX].x;
			tempSetPos[idx].y = idx;
		}
		for (idx = 0; idx<= S$THICK_MAX - idxMove; idx ++)
		{
			tempSetPos[idx].x = SetPos[idx+idxMove].x;
			tempSetPos[idx].y = idx;
		}

		memcpy(SetPos,tempSetPos,sizeof(SetPos));

	}/* if(moveValue > 0) */

	DrawMan.v1 				=  tempCurveNode[S$THICK_MAX].v1.x;
	DrawMan.v2 				=  tempCurveNode[S$THICK_MAX].v2.x;
	DrawMan.v03 			=  tempCurveNode[S$THICK_MAX].v3.x;;
	DrawMan.currentNode  	=  S$THICK_MAX;
	DrawMan.currentPoint 	=  0;
	DrawMan.flagLineFocus 	=  0;

	DrawMan.draw = 1;

}/*end of function*/

void curveClear()
{
	memset(SetPos,0,sizeof(SetPos));
	memset(CurveNode,0,sizeof(CurveNode));

	for( i = 0; i<= S$THICK_MAX; i++)
	{
	//	DrawMan.weight = 300;  //ipis0619 dont need 10% after clear
		SetPos[i].x = DrawMan.weight + 300;
		SetPos[i].y = i;
	}

	DrawMan.oldWeight 			=  DrawMan.weight;
	DrawMan.v1 						=  (DrawMan.weight + 300) + 1;
	DrawMan.v2 						=  (DrawMan.weight + 300) + 1;
	DrawMan.v03 					=  0;
	DrawMan.currentNode  	   =  S$THICK_MAX;
	DrawMan.currentPoint 		=  0;
	DrawMan.flagLineFocus 		=  0;
	CurveNode[0].former    		=  S$THICK_MAX;
	CurveNode[0].next    		=  S$THICK_MAX;
	CurveNode[0].v3.x    		=  DrawMan.weight + 300;
	CurveNode[0].v3.y    		=  0;
	CurveNode[0].flagNode  		=  1;

	CurveNode[S$THICK_MAX].former 	= 0;
	CurveNode[S$THICK_MAX].next   	= 0;
	CurveNode[S$THICK_MAX].v0.x   	= DrawMan.weight + 300;
	CurveNode[S$THICK_MAX].v0.y   	= 0;
	CurveNode[S$THICK_MAX].v3.x   	= DrawMan.weight + 300;
	CurveNode[S$THICK_MAX].v3.y   	= S$THICK_MAX;

	CurveNode[S$THICK_MAX].v1.x   	= (DrawMan.weight+ 300) + 1;
	CurveNode[S$THICK_MAX].v1.y   	= CurveNode[S$THICK_MAX].v0.y +
		(CurveNode[S$THICK_MAX].v3.y - CurveNode[S$THICK_MAX].v0.y)*1/
		3 ;
		CurveNode[S$THICK_MAX].v2.x      = (DrawMan.weight + 300) + 1;
	CurveNode[S$THICK_MAX].v2.y   	= CurveNode[S$THICK_MAX].v0.y +
		(CurveNode[S$THICK_MAX].v3.y - CurveNode[S$THICK_MAX].v0.y)*(S$THICK_V_SCALE -1)/
		S$THICK_V_SCALE;

	CurveNode[S$THICK_MAX].flagNode =  1;

	setColor = 1;
}/*end of function */
/************************************  END *******************************************/
```

#### cur_edit.var
```iecst
VAR
	x_Profile : ARRAY[0..99] OF REAL;
	TouchPoint : TouchAction;
	cntPressed : UDINT;
END_VAR
VAR RETAIN
	LengthUnit : INT;
END_VAR
VAR
	bAddLineMode : BOOL;
	IndexAddLine : UINT;
	IndexAddLineMax : UINT;
	bStartUpLineFocus : BOOL;
	bStartDnLineFocus : BOOL;
	bWeightUp : BOOL;
	bWeightDown : BOOL;
	bQuickUp : BOOL;
	bQuickDown : BOOL;
	bFocusUp : BOOL;
	bFocusDown : BOOL;
	bCurveChangeLine : BOOL;
	bCurveUpLeft : BOOL;
	bCurveUpRight : BOOL;
	bCurveDnLeft : BOOL;
	bCurveDnRight : BOOL;
	cntPressbuttonTime : UDINT;
	bCurveInit : BOOL;
	oldSetPos : ARRAY[0..399] OF position_typ;
	R_TRIG_Change : R_TRIG;
	F_TRIG_TAB : F_TRIG;
	R_TRIG_ENTER : R_TRIG;
	R_TRIG_DEL : R_TRIG;
	R_TRIG_UP : R_TRIG;
	R_TRIG_DOWN : R_TRIG;
	R_TRIG_QUICK_UP : R_TRIG;
	R_TRIG_QUICK_DOWN : R_TRIG;
	R_TRIG_CURTOL : R_TRIG;
	R_TRIG_DOWNLOAD : R_TRIG;
	R_TRIG_CLEAR : R_TRIG;
	weightUpButton : USINT;
	weightDownButton : USINT;
	quickUpButton : USINT;
	quickDownButton : USINT;
	focusUpButton : USINT;
	focusDownButton : USINT;
	tabButton : USINT;
	delButton : USINT;
	upButton : USINT;
	downButton : USINT;
	downloadButton : USINT;
	changeButton : USINT;
	curtolButton : USINT;
	escButton : USINT;
	clearButton : USINT;
	v1Add : USINT;
	v1Sub : USINT;
	v2Add : USINT;
	v2Sub : USINT;
	v03Add : USINT;
	v03Sub : USINT;
	addNode : USINT;
	delNode : USINT;
	scanNode : SINT;
	scanLine : SINT;
	curveToL : SINT;
	movePoint : SINT;
	counter0 : INT;
	counter1 : INT;
	cntTime0 : INT;
	focusColor : UINT;
	unfocusColor : UINT;
	i : UINT;
	weightStep : UINT;
	isDownLoad : USINT;
	currentGap : UINT;
	currentIndex : UINT;
	inputLock : ARRAY[0..9] OF USINT;
	Counter : UINT;
	AccuColor : UINT;
	ContiColor : UINT;
	CurevInitDownload : USINT;
	inputenable : USINT;
	inputok : USINT;
	tempGap : INT;
	oldcurrentGap : INT;
	tempCurveNode : ARRAY[0..399] OF curveNode_typ;
	tempSetPos : ARRAY[0..399] OF position_typ;
	moveInputEnable : USINT;
	moveInputOk : USINT;
	moveValue : SINT;
	nodeIdxInc : INT;
	endIdx : INT;
	startIdx : INT;
	TimeLenth : INT;
	StepLength : INT;
	RTInfo_v : RTInfo;
	tTask : REAL;
	cntUpButtonPress : UDINT;
	cntDownButtonPress : UDINT;
	cntQuickUpPress : UDINT;
	cntQuickDownPress : UDINT;
	cntFocusUpPress : UDINT;
	cntFocusDownPress : UDINT;
	mDrawMan : drawMan_typ;
	mCurveNode : ARRAY[0..399] OF curveNode_typ;
	mSetPos : ARRAY[0..399] OF position_typ;
	bKeyBack : BOOL;
	bBackEnable : BOOL;
	redoDrawMan : drawMan_typ;
	redoCurveNode : ARRAY[0..399] OF curveNode_typ;
	redoSetPos : ARRAY[0..399] OF position_typ;
	bKeyRedo : BOOL;
	bRedoEnable : BOOL;
	tempIndex : UINT;
	bHideCrossImply : UINT;
	bHideInsert : UINT;
	bHideCurveOperate : UINT;
	bHideDel : UINT;
	bHideBack : UINT;
	cntFlash : UINT;
	loadBmpGrpFlash : UINT;
	MarkPercent : INT;
	IsMarkerOld : ARRAY[0..99] OF USINT;
	GetPictureOld : UINT;
	MarkPercentOld : INT;
	ServoMinOld : INT;
	ServoMaxOld : INT;
	IsZeroDnOld : INT;
END_VAR
```

### Program Logical/thickness/exchange (ANSIC, version 1.00.0) - set thick parameter

#### exchange.c
```c
/********************************************************************
 * COPYRIGHT --  B&R Automation China
 ********************************************************************
 * Program: exchange
 * File: exchange.c
 * Author: lijianjun
 * Created: March 06, 2013
 ********************************************************************
 * Implementation of program exchangel --- data exchange control
 ********************************************************************/

#include <bur/plctypes.h>

#ifdef _DEFAULT_INCLUDES
	#include <AsDefault.h>
#endif

#define TIME_OF_CYCLE               2

/************************************************************************************
****	        		I N I T U P  O F   T H E   T A S K 		 				 ****
************************************************************************************/

void _INIT Exchange_init(void)
{
	IsAccuReCal  = 0;
	OldAccuStart = 0;
	OldAccuStop  = 0;

	gThickProf.ShareSet.OpenGapTime  = 5;
	gThickProf.ShareSet.SealGapTime  = 5;

   GapMaxLimitChange = 0;
}

/************************************************************************************
****				C Y C L I C   P A R T   O F   T H E   T A S K  				 ****
************************************************************************************/

void _CYCLIC Exchange_cyclic (void)
{
	int i;

	/* 非储料缸吹瓶机 */
	gThickProf.FunOption.IsAccu = 0;

	/* 储料缸电子尺显示 */
	if((gAccuLinear.MaxPos > gAccuLinear.ZeroPos + 1000)&&(gAccuLinear.MaxPos != 32767)&&(gAccuLinear.ZeroPos != 0))
	{
		gAccuLinear.IsReady = 1;
	}
	else
	{
		gAccuLinear.IsReady = 0;
	}

	gAccuLinear.Status      = gAccuLinear.IsReady;
	gAccuLinear.MoveLength  = (gAccuLinear.MaxPos - gAccuLinear.ZeroPos)* gAccuLinear.Length/32767;
	gAccuLinear.Unit        = gAccuLinear.Length ;
	gAccuLinear.MoveLengthV = gAccuLinear.MaxPos - gAccuLinear.ZeroPos;

	/*Albert make connect*/
	gThickData.IsZeroDn = gThickProf.FunOption.IsZeroDn;

	/* 伺服电子尺显示 */
	gServoLinear.MoveLength = (gServoLinear.MaxPos - gServoLinear.ZeroPos)* gServoLinear.Length/32767;
	gServoLinear.Unit = gServoLinear.Length;
	gServoLinear.MoveLengthV = gServoLinear.MaxPos - gServoLinear.ZeroPos;

	/* 壁厚图形改变 */
   if(gServoLinear.GapMaxLimit < 10)gServoLinear.GapMaxLimit  = 10;
   if(gServoLinear.GapMaxLimit > 100)gServoLinear.GapMaxLimit = 100;

	if(1 == gRecipeOperate.OnceOk && 1 == gRecipeOperate.CurveOk)
	{
		if(gServoLinear.GapMaxLimit != GapMaxLimitOld)
		{
			GapMaxLimitChange = 1;
		}
	}
   GapMaxLimitOld = gServoLinear.GapMaxLimit;

	//   gThickData.ServoMin = gServoLinear.ZeroPos;
	//   gThickData.ServoMax = gServoLinear.ZeroPos + (gServoLinear.MaxPos - gServoLinear.ZeroPos) * gServoLinear.GapMaxLimit /100;

	if(0 == gThickProf.FunOption.IsZeroDn)
	{
		gThickData.ServoMin = gServoLinear.ZeroPos;
		gThickData.ServoMax = gServoLinear.ZeroPos + (gServoLinear.MaxPos - gServoLinear.ZeroPos) * gServoLinear.GapMaxLimit /100;
	}
	else
	{
		gThickData.ServoMin = gServoLinear.MaxPos - (gServoLinear.MaxPos - gServoLinear.ZeroPos) * gServoLinear.GapMaxLimit /100;
		gThickData.ServoMax = gServoLinear.MaxPos;
	}

	gThickData.ServoLength = gThickData.ServoMax - gThickData.ServoMin;

	/* 封口位置 */
	if(1 == gThickProf.FunOption.SealMode)
	{
	//	if(gThickProf.ShareSet.SealGap <= 100)gThickProf.ShareSet.SealGap = 100;
		if(gThickProf.ShareSet.SealGap <= 0)gThickProf.ShareSet.SealGap = 0;   //ipis0718
	}

//	if(gThickProf.TimSet.PurgeGap < 100)gThickProf.TimSet.PurgeGap = 100;		// 2018.07.12 Jack: Remove protection

	//	gThickData.SealPos  = gThickData.ServoMin + (gThickData.ServoMax - gThickData.ServoMin)* gThickProf.ShareSet.SealGap/1000;
	//	gThickData.PurgePos = gThickData.ServoMin + (gThickData.ServoMax - gThickData.ServoMin)* gThickProf.TimSet.PurgeGap/1000;
	if(0 == gThickProf.FunOption.IsZeroDn)
	{
		gThickData.SealPos  = gThickData.ServoMin + (gThickData.ServoMax - gThickData.ServoMin)* gThickProf.ShareSet.SealGap/1000;
		gThickData.PurgePos = gThickData.ServoMin + (gThickData.ServoMax - gThickData.ServoMin)* gThickProf.TimSet.PurgeGap/1000;
	}
	else
	{
		gThickData.SealPos  = gThickData.ServoMax - (gThickData.ServoMax - gThickData.ServoMin)* gThickProf.ShareSet.SealGap/1000;
		gThickData.PurgePos = gThickData.ServoMax - (gThickData.ServoMax - gThickData.ServoMin)* gThickProf.TimSet.PurgeGap/1000;
	}

	if(gThickProf.AccuSet.StartSize != OldAccuStart)
	{
		OldAccuStart = gThickProf.AccuSet.StartSize;
		IsAccuReCal  = 1;
	}

	if(gThickProf.AccuSet.StopBuffer != OldAccuStop)
	{
		OldAccuStart = gThickProf.AccuSet.StopBuffer;
		IsAccuReCal  = 1;
	}

	/* 储料缸每点位置计算 */
	if(1 == gAccuLinear.IsReady)
	{
		if( 1 == IsAccuReCal)
		{
			gThickData.PosData[0]  = (short)(gAccuLinear.ZeroPos + (gAccuLinear.MaxPos - gAccuLinear.ZeroPos)
									        * gThickProf.AccuSet.StartSize/1000);
			gThickData.PosData[100]= (short)(gAccuLinear.ZeroPos + (gAccuLinear.MaxPos - gAccuLinear.ZeroPos)
									        * gThickProf.AccuSet.StopBuffer/1000);
			gThickData.PointLength = (gThickData.PosData[0]- gThickData.PosData[100])/100;

			for(i=1;i<100;i++)
			{
				gThickData.PosData[i] = gThickData.PosData[100] + (100 - i)*gThickData.PointLength;
			}
			IsAccuReCal = 0;
		}
		if(gThickProf.AccuSet.StartDly<= 0)gThickProf.AccuSet.StartDly = 0;
		if(gAccuLinear.Current > gThickData.PosData[0]+ gThickData.PointLength * gThickProf.AccuSet.StartDly/10)
		{
			gThickIO.Out.FullPos  = 1;
			gThickIO.Out.EmptyPos = 0;
		}
		else if(gAccuLinear.Current < gThickData.PosData[100])
		{
			gThickIO.Out.FullPos  = 0;
			gThickIO.Out.EmptyPos = 1;
		}
		else
		{
			gThickIO.Out.FullPos  = 0;
			gThickIO.Out.EmptyPos = 0;
		}

		gControlInfo.CurrentAccuPercent = (gAccuLinear.Current - gAccuLinear.ZeroPos)* 100.0 /
										          (gAccuLinear.MaxPos - gAccuLinear.ZeroPos);
	}

	/* 储料缸射出位置限制 */
	if(gThickProf.AccuSet.StartSize < 50)gThickProf.AccuSet.StartSize = 50;

	if(gThickProf.AccuSet.StartSize < gThickProf.AccuSet.StopBuffer)gThickProf.AccuSet.StopBuffer = 0;
	/* 储料当前位置显示 */
	if((1 == gAccuLinear.IsReady) && (gThickProf.AccuSet.StartSize > gThickProf.AccuSet.StopBuffer))
	{
		if(gAccuLinear.Current <= gThickData.PosData[100])
		{
			gControlInfo.CurrentAccu = 0;
		}
		else
		{
			if(gThickData.PointLength != 0)
			{
				gControlInfo.CurrentAccu = (gAccuLinear.Current - gThickData.PosData[100])* 10/gThickData.PointLength;
			}
		    if(gControlInfo.CurrentAccu > 1000 )gControlInfo.CurrentAccu = 1000;
		}
	}
	BarAccuDis = gControlInfo.CurrentAccu/10;

	/* 伺服参数传递 */
	gThickData.CycleTimes = gThickProf.TimSet.CycleTime * 5;
	if(gThickData.CycleTimes < 500)gThickData.CycleTimes = 500;

	if(gThickProf.ShareSet.OpenGapTime == 0)gThickProf.ShareSet.OpenGapTime = 5;
	if(gThickProf.ShareSet.SealGapTime == 0)gThickProf.ShareSet.SealGapTime = 5;

	gThickProf.TimSet.StartDly =0; //ipis0801
	if(0 == gThickProf.FunOption.IsAccu)
	{
		gThickData.TimeOpenDly = gThickProf.TimSet.StartDly * gThickProf.TimSet.CycleTime / 200;
	}
	else
	{
		gThickData.AccuOpenDly = gThickProf.ShareSet.OpenGapTime * 100/TIME_OF_CYCLE;
	}

	gThickData.TimePerDot = gThickData.CycleTimes/100;

	if(gThickProf.ShareSet.SealGapTime != 0)
	{
		gThickData.SealGapDly = gThickProf.ShareSet.SealGapTime * 100/TIME_OF_CYCLE;
	}
	else
	{
		gThickProf.ShareSet.SealGapTime = 5;
	}

	if(gThickProf.ShareSet.Gain >10)gThickProf.ShareSet.Gain =10;

	TimePid.KpGain = 10 + gThickProf.ShareSet.Gain * 10;

	AccuPid.KpGain = TimePid.KpGain;
	AccuPid.KdGain = TimePid.KdGain;

	if(TimePid.Wave == 0)TimePid.Wave = 10;
	AccuPid.Wave = TimePid.Wave;

	AccuPid.Change = TimePid.Change;

	if(TimePid.Slew < 200)TimePid.Slew = 200;
	AccuPid.Slew = TimePid.Slew ;

	AccuPid.RepairOut = TimePid.RepairOut;

	if(gThickProf.ShareSet.MarkerTime < 1)gThickProf.ShareSet.MarkerTime = 5;

	if(gThickProf.ShareSet.ThickFlow < 200)gThickProf.ShareSet.ThickFlow = 800;
	if(gThickProf.ShareSet.StartFlow < 200)gThickProf.ShareSet.StartFlow = 700;
	if(gThickProf.ShareSet.SealFlow < 200 )gThickProf.ShareSet.SealFlow  = 700;

	/*gImply.ParisonPumpNotOn = !gServoLinear.IsReady;*/
}/* cyclic part end  */
```

#### exchange.var
```iecst
VAR
	OldAccuStart : UINT;
	OldAccuStop : UINT;
	IsAccuReCal : USINT;
	GapMaxLimitOld : REAL;
	BarAccuDis : USINT;
END_VAR
```

### Program Logical/thickness/cur_save (ANSIC, version 1.00.0) - profile save

#### cur_save.typ - Local data types
```iecst
(********************************************************************
 * COPYRIGHT --  B&R CHINA
 ********************************************************************
 * Program: cur_save
 * File: cur_save.typ
 * Author: lij
 * Created: March 06, 2013
 ********************************************************************
 * Local data types of program cur_save --- thickness profile load/save
 ********************************************************************)

TYPE
	curveData_typ : 	STRUCT
		CurveNode : ARRAY[0..399]OF curveNode_typ;
		SetPos : ARRAY[0..399]OF position_typ;
		weight : INT;
		v1 : INT;
		v2 : INT;
		v03 : INT;
		currentPoint : INT;
		currentNode : INT;
		usedIndex : UINT;
		flagLineFocus : USINT;
	END_STRUCT;
END_TYPE
```

#### cur_save.var
```iecst
VAR
	DataObjOperate : DatObj_Operate_typ;
	indexRecipe : UINT;
	DatObj_Info : DatObjInfo;
	DatObj_Create : DatObjCreate;
	DatObj_Write : DatObjWrite;
	DatObj_Read : DatObjRead;
	i : UINT;
	counter : UINT;
	curveIndex : UINT;
	curveIndexOld : UINT;
	curveData : ARRAY[0..4] OF curveData_typ;
	status_tmpalloc : UINT;
	status_tmpfree : UINT;
	pCurveData : UDINT;
	fileSingleName : STRING[80];
	fileAllName : STRING[80];
	FileOpen_0 : FileOpen;
	FileCreate_0 : FileCreate;
	FileWrite_0 : FileWrite;
	FileRead_0 : FileRead;
	FileClose_0 : FileClose;
END_VAR
```
